KUKA KRL program: EPS_2_251825_SA36_A_20260116064122.src

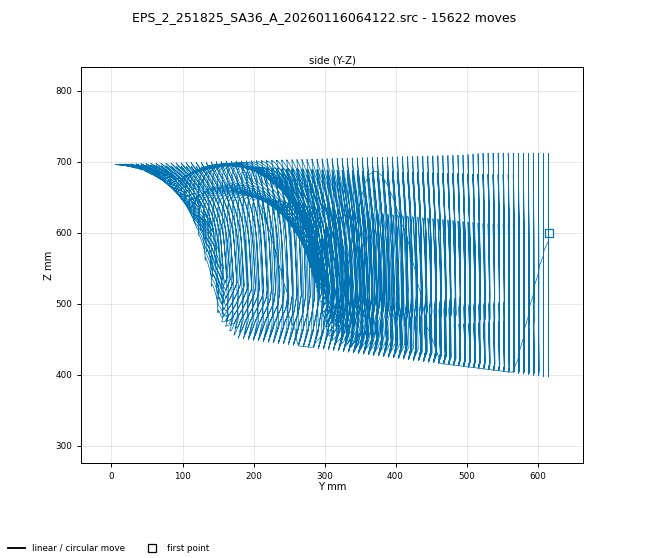
[picture p0: tool path of EPS_2_251825_SA36_A_20260116064122.src, 15622 of 15624 moves have a stored position in this frame; points joined in program order, loops and branches not executed]
&ACCESS RVP
&REL 4
&COMMENT QRS 19112012
&PARAM EDITMASK = *
DEF PART()
EXT BAS (BAS_COMMAND :IN,REAL :IN )
INT I
BAS (#INITMOV,0 )

;KUKA QRS Post kuka4.cps  Date:22-06-2017 !

File_ID=2974

QRS_PRE_INIT()

;Init var - Until changes are made in qrs_pre_init
Outlet_Square_prg=0
Inlet_1_Square_prg=0
Inlet_2_Square_prg=0
Inlet_3_Square_prg=0
Inlet_4_Square_prg=0
Inlet_5_Square_prg=0

Outlet_1={X 0.000, Y 524.580, Z 611.500, B 0.000, E1 0.000 }
Inlet_1={X 0.000, Y 531.710, Z 511.500, B 0.000, E1 90.000 }
Inlet_2={X 0.000, Y 526.720, Z 581.500, B 0.000, E1 180.000 }
Inlet_3={X 0.000, Y 526.720, Z 581.500, B 0.000, E1 270.000 }
Outlet_1_type=201
Inlet_1_type=201
Inlet_2_type=201
Inlet_3_type=201
;QRS#1=Sidecore dimensions
;QRS#2=200-8" PVC SDR 35
;QRS#3=200-8" PVC SDR 35
;QRS#4=200-8" PVC SDR 35
;QRS#5=200-8" PVC SDR 35
;QRS#6=
;QRS#7=
;QRS#8=
;QRS#9=12-08 PSX
;QRS#10=12-08 PSX
;QRS#11=12-08 PSX
;QRS#12=12-08 PSX
;QRS#13=
;QRS#14=
;QRS#15=
;QRS#16=1220x127x991 3,25'
;QRS#17=EPS Height
;QRS#18=712
;QRS#19=*
;QRS#20= UPDATED VERSION 22-06-2017
;QRS#21=*
Outlet_Square=0100
Inlet_1_Square=0100
Inlet_2_Square=0100
Inlet_3_Square=0100
Inlet_4_Square=0
Inlet_5_Square=0
Mill_Square=1
Outlet_Square_Prg=204
Inlet_1_Square_prg=204
Inlet_2_Square_prg=204
Inlet_3_Square_prg=204

QRS_INIT()

$ADVANCE=5

; T1
PTP {E1 173.498,E2 173.498}
PTP {X 0,Y 615.498,A -85,B 0,C 180,E1 173.498,E2 173.498,E3 0,E4 0,E5 0,E6 0}
QRS_SPEED_INIT()
LIN {X 0,Y 615.498,Z 600,A -85,B 0,C 180,E1 173.498,E2 173.498,E3 0,E4 0,E5 0,E6 0} C_VEL
LIN {X 0,Y 615.498,Z 591.852,A -85,B 0,C 180,E1 173.498,E2 173.498} C_VEL
LIN {X 0,Y 615.496,Z 590.208,A -85,B 0,C 180,E1 173.418,E2 173.418} C_VEL
LIN {X 0,Y 615.497,Z 582.536,A -85,B 0,C 180,E1 172.455,E2 172.455} C_VEL
LIN {X 0,Y 615.498,Z 572.758,A -85,B 0,C 180,E1 171.463,E2 171.463} C_VEL
LIN {X 0,Y 615.498,Z 562.492,A -85,B 0,C 180,E1 170.636,E2 170.636} C_VEL
LIN {X 0,Y 615.491,Z 550.929,A -85,B 0,C 180,E1 169.889,E2 169.889} C_VEL
LIN {X 0,Y 615.495,Z 539.071,A -85,B 0,C 180,E1 169.293,E2 169.293} C_VEL
LIN {X 0,Y 615.478,Z 526.159,A -85,B 0,C 180,E1 168.807,E2 168.807} C_VEL
LIN {X 0,Y 615.485,Z 513.556,A -85,B 0,C 180,E1 168.473,E2 168.473} C_VEL
LIN {X 0,Y 615.495,Z 500.425,A -85,B 0,C 180,E1 168.265,E2 168.265} C_VEL
LIN {X 0,Y 615.485,Z 402.646,A -85,B 0,C 180,E1 167.113,E2 167.113} C_VEL
LIN {X 0,Y 615.478,Z 396.69,A -85,B 0,C 180,E1 165.834,E2 165.834} C_VEL
LIN {X 0,Y 615.447,Z 396.692,A -85,B 0,C 180,E1 163.412,E2 163.412} C_VEL
LIN {X 0,Y 615.448,Z 396.692,A -85,B 0,C 180,E1 161.353,E2 161.353} C_VEL
LIN {X 0,Y 615.498,Z 396.7,A -85,B 0,C 180,E1 158.568,E2 158.568} C_VEL
LIN {X 0,Y 615.473,Z 396.686,A -85,B 0,C 180,E1 155.727,E2 155.727} C_VEL
LIN {X 0,Y 615.476,Z 396.697,A -85,B 0,C 180,E1 152.958,E2 152.958} C_VEL
LIN {X 0,Y 615.489,Z 396.686,A -85,B 0,C 180,E1 150.206,E2 150.206} C_VEL
LIN {X 0,Y 615.471,Z 396.688,A -85,B 0,C 180,E1 147.541,E2 147.541} C_VEL
LIN {X 0,Y 615.476,Z 396.696,A -85,B 0,C 180,E1 145.184,E2 145.184} C_VEL
LIN {X 0,Y 615.485,Z 396.696,A -85,B 0,C 180,E1 142.757,E2 142.757} C_VEL
LIN {X 0,Y 615.493,Z 396.682,A -85,B 0,C 180,E1 139.911,E2 139.911} C_VEL
LIN {X 0,Y 615.484,Z 396.697,A -85,B 0,C 180,E1 136.953,E2 136.953} C_VEL
LIN {X 0,Y 615.487,Z 396.684,A -85,B 0,C 180,E1 133.997,E2 133.997} C_VEL
LIN {X 0,Y 615.477,Z 396.698,A -85,B 0,C 180,E1 131.093,E2 131.093} C_VEL
LIN {X 0,Y 615.463,Z 396.694,A -85,B 0,C 180,E1 128.906,E2 128.906} C_VEL
LIN {X 0,Y 615.461,Z 396.689,A -85,B 0,C 180,E1 126.427,E2 126.427} C_VEL
LIN {X 0,Y 615.498,Z 396.699,A -85,B 0,C 180,E1 123.535,E2 123.535} C_VEL
LIN {X 0,Y 615.445,Z 396.695,A -85,B 0,C 180,E1 120.922,E2 120.922} C_VEL
LIN {X 0,Y 615.452,Z 396.692,A -85,B 0,C 180,E1 118.444,E2 118.444} C_VEL
LIN {X 0,Y 615.477,Z 396.7,A -85,B 0,C 180,E1 115.566,E2 115.566} C_VEL
LIN {X 0,Y 615.47,Z 396.699,A -85,B 0,C 180,E1 113.557,E2 113.557} C_VEL
LIN {X 0,Y 615.44,Z 396.801,A -85,B 0,C 180,E1 112.513,E2 112.513} C_VEL
LIN {X 0,Y 615.481,Z 417.648,A -85,B 0,C 180,E1 109.685,E2 109.685} C_VEL
LIN {X 0,Y 615.457,Z 437.029,A -85,B 0,C 180,E1 107.1,E2 107.1} C_VEL
LIN {X 0,Y 615.482,Z 457.56,A -85,B 0,C 180,E1 104.396,E2 104.396} C_VEL
LIN {X 0,Y 615.455,Z 469.845,A -85,B 0,C 180,E1 102.824,E2 102.824} C_VEL
LIN {X 0,Y 615.464,Z 577.646,A -85,B 0,C 180,E1 101.548,E2 101.548} C_VEL
LIN {X 0,Y 615.46,Z 590.227,A -85,B 0,C 180,E1 101.277,E2 101.277} C_VEL
LIN {X 0,Y 615.48,Z 602.525,A -85,B 0,C 180,E1 100.883,E2 100.883} C_VEL
LIN {X 0,Y 615.489,Z 614.565,A -85,B 0,C 180,E1 100.361,E2 100.361} C_VEL
LIN {X 0,Y 615.491,Z 626.304,A -85,B 0,C 180,E1 99.696,E2 99.696} C_VEL
LIN {X 0,Y 615.499,Z 636.767,A -85,B 0,C 180,E1 98.95,E2 98.95} C_VEL
LIN {X 0,Y 615.498,Z 645.33,A -85,B 0,C 180,E1 98.206,E2 98.206} C_VEL
LIN {X 0,Y 615.497,Z 653.209,A -85,B 0,C 180,E1 97.38,E2 97.38} C_VEL
LIN {X 0,Y 615.497,Z 660.898,A -85,B 0,C 180,E1 96.392,E2 96.392} C_VEL
LIN {X 0,Y 615.497,Z 667.958,A -85,B 0,C 180,E1 95.241,E2 95.241} C_VEL
LIN {X 0,Y 615.494,Z 672.658,A -85,B 0,C 180,E1 94.256,E2 94.256} C_VEL
LIN {X 0,Y 615.494,Z 676.254,A -85,B 0,C 180,E1 93.273,E2 93.273} C_VEL
LIN {X 0,Y 615.496,Z 678.115,A -85,B 0,C 180,E1 92.618,E2 92.618} C_VEL
LIN {X 0,Y 615.499,Z 679.533,A -85,B 0,C 180,E1 91.963,E2 91.963} C_VEL
LIN {X 0,Y 615.496,Z 681.141,A -85,B 0,C 180,E1 90.654,E2 90.654} C_VEL
LIN {X 0,Y 615.495,Z 681.384,A -85,B 0,C 180,E1 90,E2 90} C_VEL
LIN {X 0,Y 615.495,Z 681.206,A -85,B 0,C 180,E1 89.346,E2 89.346} C_VEL
LIN {X 0,Y 615.499,Z 679.682,A -85,B 0,C 180,E1 88.037,E2 88.037} C_VEL
LIN {X 0,Y 615.498,Z 678.341,A -85,B 0,C 180,E1 87.382,E2 87.382} C_VEL
LIN {X 0,Y 615.496,Z 675.494,A -85,B 0,C 180,E1 86.399,E2 86.399} C_VEL
LIN {X 0,Y 615.498,Z 671.634,A -85,B 0,C 180,E1 85.416,E2 85.416} C_VEL
LIN {X 0,Y 615.498,Z 666.651,A -85,B 0,C 180,E1 84.43,E2 84.43} C_VEL
LIN {X 0,Y 615.496,Z 660.208,A -85,B 0,C 180,E1 83.418,E2 83.418} C_VEL
LIN {X 0,Y 615.497,Z 652.536,A -85,B 0,C 180,E1 82.455,E2 82.455} C_VEL
LIN {X 0,Y 615.498,Z 642.758,A -85,B 0,C 180,E1 81.463,E2 81.463} C_VEL
LIN {X 0,Y 615.498,Z 632.492,A -85,B 0,C 180,E1 80.636,E2 80.636} C_VEL
LIN {X 0,Y 615.491,Z 620.929,A -85,B 0,C 180,E1 79.889,E2 79.889} C_VEL
LIN {X 0,Y 615.495,Z 609.089,A -85,B 0,C 180,E1 79.294,E2 79.294} C_VEL
LIN {X 0,Y 615.467,Z 596.161,A -85,B 0,C 180,E1 78.806,E2 78.806} C_VEL
LIN {X 0,Y 615.466,Z 583.56,A -85,B 0,C 180,E1 78.473,E2 78.473} C_VEL
LIN {X 0,Y 615.476,Z 570.434,A -85,B 0,C 180,E1 78.264,E2 78.264} C_VEL
LIN {X 0,Y 615.455,Z 469.493,A -85,B 0,C 180,E1 77.071,E2 77.071} C_VEL
LIN {X 0,Y 615.473,Z 449.33,A -85,B 0,C 180,E1 74.434,E2 74.434} C_VEL
LIN {X 0,Y 615.472,Z 427.636,A -85,B 0,C 180,E1 71.562,E2 71.562} C_VEL
LIN {X 0,Y 615.457,Z 407.969,A -85,B 0,C 180,E1 68.918,E2 68.918} C_VEL
LIN {X 0,Y 615.43,Z 396.698,A -85,B 0,C 180,E1 67.376,E2 67.376} C_VEL
LIN {X 0,Y 615.429,Z 396.697,A -85,B 0,C 180,E1 65.006,E2 65.006} C_VEL
LIN {X 0,Y 615.491,Z 396.694,A -85,B 0,C 180,E1 62.085,E2 62.085} C_VEL
LIN {X 0,Y 615.479,Z 396.689,A -85,B 0,C 180,E1 59.839,E2 59.839} C_VEL
LIN {X 0,Y 615.457,Z 396.69,A -85,B 0,C 180,E1 57.541,E2 57.541} C_VEL
LIN {X 0,Y 615.455,Z 396.694,A -85,B 0,C 180,E1 55.183,E2 55.183} C_VEL
LIN {X 0,Y 615.481,Z 396.701,A -85,B 0,C 180,E1 52.757,E2 52.757} C_VEL
LIN {X 0,Y 615.491,Z 396.683,A -85,B 0,C 180,E1 49.911,E2 49.911} C_VEL
LIN {X 0,Y 615.475,Z 396.687,A -85,B 0,C 180,E1 47.646,E2 47.646} C_VEL
LIN {X 0,Y 615.496,Z 396.7,A -85,B 0,C 180,E1 44.932,E2 44.932} C_VEL
LIN {X 0,Y 615.49,Z 396.683,A -85,B 0,C 180,E1 42.08,E2 42.08} C_VEL
LIN {X 0,Y 615.489,Z 396.698,A -85,B 0,C 180,E1 39.062,E2 39.062} C_VEL
LIN {X 0,Y 615.468,Z 396.688,A -85,B 0,C 180,E1 36.426,E2 36.426} C_VEL
LIN {X 0,Y 615.49,Z 396.697,A -85,B 0,C 180,E1 33.534,E2 33.534} C_VEL
LIN {X 0,Y 615.454,Z 396.695,A -85,B 0,C 180,E1 30.922,E2 30.922} C_VEL
LIN {X 0,Y 615.455,Z 396.691,A -85,B 0,C 180,E1 28.444,E2 28.444} C_VEL
LIN {X 0,Y 615.484,Z 396.7,A -85,B 0,C 180,E1 25.567,E2 25.567} C_VEL
LIN {X 0,Y 615.473,Z 396.699,A -85,B 0,C 180,E1 23.557,E2 23.557} C_VEL
LIN {X 0,Y 615.441,Z 396.801,A -85,B 0,C 180,E1 22.513,E2 22.513} C_VEL
LIN {X 0,Y 615.481,Z 417.648,A -85,B 0,C 180,E1 19.685,E2 19.685} C_VEL
LIN {X 0,Y 615.457,Z 437.029,A -85,B 0,C 180,E1 17.1,E2 17.1} C_VEL
LIN {X 0,Y 615.482,Z 457.56,A -85,B 0,C 180,E1 14.396,E2 14.396} C_VEL
LIN {X 0,Y 615.455,Z 469.843,A -85,B 0,C 180,E1 12.824,E2 12.824} C_VEL
LIN {X 0,Y 615.464,Z 577.645,A -85,B 0,C 180,E1 11.548,E2 11.548} C_VEL
LIN {X 0,Y 615.46,Z 590.226,A -85,B 0,C 180,E1 11.277,E2 11.277} C_VEL
LIN {X 0,Y 615.48,Z 602.525,A -85,B 0,C 180,E1 10.883,E2 10.883} C_VEL
LIN {X 0,Y 615.489,Z 614.564,A -85,B 0,C 180,E1 10.361,E2 10.361} C_VEL
LIN {X 0,Y 615.491,Z 626.303,A -85,B 0,C 180,E1 9.696,E2 9.696} C_VEL
LIN {X 0,Y 615.499,Z 636.767,A -85,B 0,C 180,E1 8.95,E2 8.95} C_VEL
LIN {X 0,Y 615.498,Z 645.33,A -85,B 0,C 180,E1 8.206,E2 8.206} C_VEL
LIN {X 0,Y 615.497,Z 653.209,A -85,B 0,C 180,E1 7.381,E2 7.381} C_VEL
LIN {X 0,Y 615.497,Z 660.898,A -85,B 0,C 180,E1 6.392,E2 6.392} C_VEL
LIN {X 0,Y 615.497,Z 667.958,A -85,B 0,C 180,E1 5.241,E2 5.241} C_VEL
LIN {X 0,Y 615.494,Z 672.658,A -85,B 0,C 180,E1 4.256,E2 4.256} C_VEL
LIN {X 0,Y 615.494,Z 676.254,A -85,B 0,C 180,E1 3.273,E2 3.273} C_VEL
LIN {X 0,Y 615.496,Z 678.115,A -85,B 0,C 180,E1 2.618,E2 2.618} C_VEL
LIN {X 0,Y 615.499,Z 679.533,A -85,B 0,C 180,E1 1.963,E2 1.963} C_VEL
LIN {X 0,Y 615.496,Z 681.141,A -85,B 0,C 180,E1 0.654,E2 0.654} C_VEL
LIN {X 0,Y 615.495,Z 681.384,A -85,B 0,C 180,E1 0,E2 0} C_VEL
LIN {X 0,Y 615.495,Z 681.206,A -85,B 0,C 180,E1 -0.654,E2 -0.654} C_VEL
LIN {X 0,Y 615.499,Z 679.682,A -85,B 0,C 180,E1 -1.963,E2 -1.963} C_VEL
LIN {X 0,Y 615.498,Z 678.341,A -85,B 0,C 180,E1 -2.618,E2 -2.618} C_VEL
LIN {X 0,Y 615.496,Z 675.494,A -85,B 0,C 180,E1 -3.601,E2 -3.601} C_VEL
LIN {X 0,Y 615.498,Z 671.634,A -85,B 0,C 180,E1 -4.584,E2 -4.584} C_VEL
LIN {X 0,Y 615.498,Z 666.651,A -85,B 0,C 180,E1 -5.57,E2 -5.57} C_VEL
LIN {X 0,Y 615.496,Z 660.208,A -85,B 0,C 180,E1 -6.582,E2 -6.582} C_VEL
LIN {X 0,Y 615.497,Z 652.537,A -85,B 0,C 180,E1 -7.545,E2 -7.545} C_VEL
LIN {X 0,Y 615.498,Z 642.759,A -85,B 0,C 180,E1 -8.536,E2 -8.536} C_VEL
LIN {X 0,Y 615.498,Z 632.493,A -85,B 0,C 180,E1 -9.364,E2 -9.364} C_VEL
LIN {X 0,Y 615.491,Z 620.93,A -85,B 0,C 180,E1 -10.111,E2 -10.111} C_VEL
LIN {X 0,Y 615.495,Z 609.09,A -85,B 0,C 180,E1 -10.706,E2 -10.706} C_VEL
LIN {X 0,Y 615.467,Z 596.163,A -85,B 0,C 180,E1 -11.193,E2 -11.193} C_VEL
LIN {X 0,Y 615.466,Z 583.562,A -85,B 0,C 180,E1 -11.527,E2 -11.527} C_VEL
LIN {X 0,Y 615.476,Z 570.437,A -85,B 0,C 180,E1 -11.736,E2 -11.736} C_VEL
LIN {X 0,Y 615.455,Z 469.493,A -85,B 0,C 180,E1 -12.929,E2 -12.929} C_VEL
LIN {X 0,Y 615.473,Z 449.33,A -85,B 0,C 180,E1 -15.566,E2 -15.566} C_VEL
LIN {X 0,Y 615.472,Z 427.636,A -85,B 0,C 180,E1 -18.438,E2 -18.438} C_VEL
LIN {X 0,Y 615.457,Z 407.969,A -85,B 0,C 180,E1 -21.082,E2 -21.082} C_VEL
LIN {X 0,Y 615.43,Z 396.698,A -85,B 0,C 180,E1 -22.624,E2 -22.624} C_VEL
LIN {X 0,Y 615.429,Z 396.697,A -85,B 0,C 180,E1 -24.994,E2 -24.994} C_VEL
LIN {X 0,Y 615.491,Z 396.694,A -85,B 0,C 180,E1 -27.915,E2 -27.915} C_VEL
LIN {X 0,Y 615.48,Z 396.689,A -85,B 0,C 180,E1 -30.161,E2 -30.161} C_VEL
LIN {X 0,Y 615.457,Z 396.69,A -85,B 0,C 180,E1 -32.459,E2 -32.459} C_VEL
LIN {X 0,Y 615.457,Z 396.694,A -85,B 0,C 180,E1 -34.817,E2 -34.817} C_VEL
LIN {X 0,Y 615.486,Z 396.701,A -85,B 0,C 180,E1 -37.242,E2 -37.242} C_VEL
LIN {X 0,Y 615.491,Z 396.683,A -85,B 0,C 180,E1 -40.089,E2 -40.089} C_VEL
LIN {X 0,Y 615.486,Z 396.702,A -85,B 0,C 180,E1 -43.047,E2 -43.047} C_VEL
LIN {X 0,Y 615.487,Z 396.683,A -85,B 0,C 180,E1 -46.003,E2 -46.003} C_VEL
LIN {X 0,Y 615.485,Z 396.702,A -85,B 0,C 180,E1 -48.906,E2 -48.906} C_VEL
LIN {X 0,Y 615.474,Z 396.695,A -85,B 0,C 180,E1 -51.094,E2 -51.094} C_VEL
LIN {X 0,Y 615.466,Z 396.688,A -85,B 0,C 180,E1 -53.574,E2 -53.574} C_VEL
LIN {X 0,Y 615.495,Z 396.697,A -85,B 0,C 180,E1 -56.465,E2 -56.465} C_VEL
LIN {X 0,Y 615.449,Z 396.695,A -85,B 0,C 180,E1 -59.078,E2 -59.078} C_VEL
LIN {X 0,Y 615.453,Z 396.692,A -85,B 0,C 180,E1 -61.556,E2 -61.556} C_VEL
LIN {X 0,Y 615.475,Z 396.699,A -85,B 0,C 180,E1 -64.434,E2 -64.434} C_VEL
LIN {X 0,Y 615.437,Z 396.843,A -85,B 0,C 180,E1 -65.411,E2 -65.411} C_VEL
LIN {X 0,Y 615.475,Z 420.552,A -85,B 0,C 180,E1 -68.216,E2 -68.216} C_VEL
LIN {X 0,Y 615.476,Z 443.127,A -85,B 0,C 180,E1 -70.835,E2 -70.835} C_VEL
LIN {X 0,Y 615.465,Z 467.126,A -85,B 0,C 180,E1 -73.577,E2 -73.577} C_VEL
LIN {X 0,Y 615.45,Z 492.711,A -85,B 0,C 180,E1 -76.462,E2 -76.462} C_VEL
LIN {X 0,Y 615.446,Z 498.522,A -85,B 0,C 180,E1 -77.113,E2 -77.113} C_VEL
LIN {X 0,Y 615.467,Z 607.831,A -85,B 0,C 180,E1 -78.41,E2 -78.41} C_VEL
LIN {X 0,Y 615.463,Z 620.346,A -85,B 0,C 180,E1 -78.681,E2 -78.681} C_VEL
LIN {X 0,Y 615.484,Z 633.665,A -85,B 0,C 180,E1 -79.115,E2 -79.115} C_VEL
LIN {X 0,Y 615.486,Z 645.476,A -85,B 0,C 180,E1 -79.639,E2 -79.639} C_VEL
LIN {X 0,Y 615.492,Z 656.993,A -85,B 0,C 180,E1 -80.304,E2 -80.304} C_VEL
LIN {X 0,Y 615.499,Z 667.34,A -85,B 0,C 180,E1 -81.05,E2 -81.05} C_VEL
LIN {X 0,Y 615.497,Z 675.811,A -85,B 0,C 180,E1 -81.794,E2 -81.794} C_VEL
LIN {X 0,Y 615.498,Z 683.606,A -85,B 0,C 180,E1 -82.62,E2 -82.62} C_VEL
LIN {X 0,Y 615.496,Z 691.203,A -85,B 0,C 180,E1 -83.608,E2 -83.608} C_VEL
LIN {X 0,Y 615.498,Z 698.204,A -85,B 0,C 180,E1 -84.759,E2 -84.759} C_VEL
LIN {X 0,Y 615.494,Z 702.851,A -85,B 0,C 180,E1 -85.744,E2 -85.744} C_VEL
LIN {X 0,Y 615.494,Z 706.399,A -85,B 0,C 180,E1 -86.727,E2 -86.727} C_VEL
LIN {X 0,Y 615.497,Z 708.233,A -85,B 0,C 180,E1 -87.382,E2 -87.382} C_VEL
LIN {X 0,Y 615.499,Z 709.608,A -85,B 0,C 180,E1 -88.037,E2 -88.037} C_VEL
LIN {X 0,Y 615.496,Z 711.174,A -85,B 0,C 180,E1 -89.346,E2 -89.346} C_VEL
LIN {X 0,Y 615.494,Z 711.389,A -85,B 0,C 180,E1 -90,E2 -90} C_VEL
LIN {X 0,Y 615.495,Z 710.58,A -85,B 0,C 180,E1 -91.309,E2 -91.309} C_VEL
LIN {X 0,Y 615.499,Z 709.608,A -85,B 0,C 180,E1 -91.963,E2 -91.963} C_VEL
LIN {X 0,Y 615.497,Z 708.233,A -85,B 0,C 180,E1 -92.618,E2 -92.618} C_VEL
LIN {X 0,Y 615.496,Z 705.349,A -85,B 0,C 180,E1 -93.601,E2 -93.601} C_VEL
LIN {X 0,Y 615.498,Z 701.441,A -85,B 0,C 180,E1 -94.584,E2 -94.584} C_VEL
LIN {X 0,Y 615.499,Z 696.405,A -85,B 0,C 180,E1 -95.57,E2 -95.57} C_VEL
LIN {X 0,Y 615.497,Z 689.869,A -85,B 0,C 180,E1 -96.583,E2 -96.583} C_VEL
LIN {X 0,Y 615.497,Z 682.133,A -85,B 0,C 180,E1 -97.545,E2 -97.545} C_VEL
LIN {X 0,Y 615.498,Z 674.044,A -85,B 0,C 180,E1 -98.371,E2 -98.371} C_VEL
LIN {X 0,Y 615.499,Z 664.167,A -85,B 0,C 180,E1 -99.199,E2 -99.199} C_VEL
LIN {X 0,Y 615.491,Z 652.98,A -85,B 0,C 180,E1 -99.945,E2 -99.945} C_VEL
LIN {X 0,Y 615.487,Z 642.021,A -85,B 0,C 180,E1 -100.527,E2 -100.527} C_VEL
LIN {X 0,Y 615.473,Z 629.516,A -85,B 0,C 180,E1 -101.039,E2 -101.039} C_VEL
LIN {X 0,Y 615.463,Z 617.067,A -85,B 0,C 180,E1 -101.402,E2 -101.402} C_VEL
LIN {X 0,Y 615.47,Z 603.466,A -85,B 0,C 180,E1 -101.652,E2 -101.652} C_VEL
LIN {X 0,Y 615.446,Z 498.522,A -85,B 0,C 180,E1 -102.887,E2 -102.887} C_VEL
LIN {X 0,Y 615.482,Z 474.694,A -85,B 0,C 180,E1 -105.566,E2 -105.566} C_VEL
LIN {X 0,Y 615.484,Z 450.837,A -85,B 0,C 180,E1 -108.28,E2 -108.28} C_VEL
LIN {X 0,Y 615.463,Z 428.078,A -85,B 0,C 180,E1 -110.907,E2 -110.907} C_VEL
LIN {X 0,Y 615.467,Z 405.498,A -85,B 0,C 180,E1 -113.557,E2 -113.557} C_VEL
LIN {X 0,Y 615.434,Z 396.696,A -85,B 0,C 180,E1 -114.634,E2 -114.634} C_VEL
LIN {X 0,Y 615.435,Z 396.697,A -85,B 0,C 180,E1 -117.035,E2 -117.035} C_VEL
LIN {X 0,Y 615.496,Z 396.696,A -85,B 0,C 180,E1 -119.796,E2 -119.796} C_VEL
LIN {X 0,Y 615.453,Z 396.691,A -85,B 0,C 180,E1 -122.46,E2 -122.46} C_VEL
LIN {X 0,Y 615.445,Z 396.694,A -85,B 0,C 180,E1 -124.818,E2 -124.818} C_VEL
LIN {X 0,Y 615.476,Z 396.698,A -85,B 0,C 180,E1 -127.243,E2 -127.243} C_VEL
LIN {X 0,Y 615.49,Z 396.684,A -85,B 0,C 180,E1 -130.089,E2 -130.089} C_VEL
LIN {X 0,Y 615.469,Z 396.687,A -85,B 0,C 180,E1 -132.355,E2 -132.355} C_VEL
LIN {X 0,Y 615.476,Z 396.699,A -85,B 0,C 180,E1 -135.07,E2 -135.07} C_VEL
LIN {X 0,Y 615.491,Z 396.683,A -85,B 0,C 180,E1 -137.92,E2 -137.92} C_VEL
LIN {X 0,Y 615.48,Z 396.685,A -85,B 0,C 180,E1 -140.249,E2 -140.249} C_VEL
LIN {X 0,Y 615.487,Z 396.702,A -85,B 0,C 180,E1 -143.064,E2 -143.064} C_VEL
LIN {X 0,Y 615.49,Z 396.682,A -85,B 0,C 180,E1 -145.978,E2 -145.978} C_VEL
LIN {X 0,Y 615.486,Z 396.703,A -85,B 0,C 180,E1 -148.915,E2 -148.915} C_VEL
LIN {X 0,Y 615.47,Z 396.688,A -85,B 0,C 180,E1 -151.553,E2 -151.553} C_VEL
LIN {X 0,Y 615.483,Z 396.69,A -85,B 0,C 180,E1 -154.284,E2 -154.284} C_VEL
LIN {X 0,Y 615.49,Z 396.694,A -85,B 0,C 180,E1 -156.444,E2 -156.444} C_VEL
LIN {X 0,Y 615.457,Z 396.692,A -85,B 0,C 180,E1 -159.268,E2 -159.268} C_VEL
LIN {X 0,Y 615.493,Z 396.686,A -85,B 0,C 180,E1 -162.043,E2 -162.043} C_VEL
LIN {X 0,Y 615.467,Z 396.697,A -85,B 0,C 180,E1 -164.773,E2 -164.773} C_VEL
LIN {X 0,Y 615.491,Z 396.874,A -85,B 0,C 180,E1 -165.988,E2 -165.988} C_VEL
LIN {X 0,Y 615.486,Z 402.617,A -85,B 0,C 180,E1 -167.197,E2 -167.197} C_VEL
LIN {X 0,Y 615.487,Z 508.791,A -85,B 0,C 180,E1 -168.473,E2 -168.473} C_VEL
LIN {X 0,Y 615.477,Z 521.741,A -85,B 0,C 180,E1 -168.765,E2 -168.765} C_VEL
LIN {X 0,Y 615.488,Z 533.654,A -85,B 0,C 180,E1 -169.159,E2 -169.159} C_VEL
LIN {X 0,Y 615.489,Z 546.195,A -85,B 0,C 180,E1 -169.723,E2 -169.723} C_VEL
LIN {X 0,Y 615.491,Z 557.576,A -85,B 0,C 180,E1 -170.387,E2 -170.387} C_VEL
LIN {X 0,Y 615.498,Z 567.823,A -85,B 0,C 180,E1 -171.133,E2 -171.133} C_VEL
LIN {X 0,Y 615.499,Z 577.034,A -85,B 0,C 180,E1 -171.959,E2 -171.959} C_VEL
LIN {X 0,Y 615.499,Z 585.892,A -85,B 0,C 180,E1 -172.943,E2 -172.943} C_VEL
LIN {X 0,Y 615.497,Z 593.123,A -85,B 0,C 180,E1 -173.937,E2 -173.937} C_VEL
LIN {X 0,Y 615.497,Z 597.958,A -85,B 0,C 180,E1 -174.759,E2 -174.759} C_VEL
LIN {X 0,Y 615.494,Z 602.658,A -85,B 0,C 180,E1 -175.744,E2 -175.744} C_VEL
LIN {X 0,Y 615.494,Z 606.255,A -85,B 0,C 180,E1 -176.727,E2 -176.727} C_VEL
LIN {X 0,Y 615.496,Z 608.115,A -85,B 0,C 180,E1 -177.382,E2 -177.382} C_VEL
LIN {X 0,Y 615.499,Z 609.533,A -85,B 0,C 180,E1 -178.037,E2 -178.037} C_VEL
LIN {X 0,Y 615.496,Z 611.142,A -85,B 0,C 180,E1 -179.346,E2 -179.346} C_VEL
LIN {X 0,Y 615.495,Z 611.384,A -85,B 0,C 180,E1 -180,E2 -180} C_VEL
LIN {X 0,Y 615.495,Z 611.206,A -85,B 0,C 180,E1 -180.654,E2 -180.654} C_VEL
LIN {X 0,Y 615.499,Z 609.682,A -85,B 0,C 180,E1 -181.963,E2 -181.963} C_VEL
LIN {X 0,Y 615.498,Z 608.341,A -85,B 0,C 180,E1 -182.618,E2 -182.618} C_VEL
LIN {X 0,Y 615.496,Z 605.494,A -85,B 0,C 180,E1 -183.601,E2 -183.601} C_VEL
LIN {X 0,Y 615.498,Z 601.634,A -85,B 0,C 180,E1 -184.585,E2 -184.585} C_VEL
LIN {X 0,Y 615.498,Z 596.651,A -85,B 0,C 180,E1 -185.57,E2 -185.57} C_VEL
LIN {X 0,Y 615.496,Z 590.208,A -85,B 0,C 180,E1 -186.582,E2 -186.582} C_VEL
LIN {X 0,Y 614.829,Z 587.026,A -85,B 0,C 180,E1 -187.031,E2 -187.031} C_VEL
LIN {X 0,Y 611.989,Z 581.452,A -85,B 0,C 180,E1 -187.748,E2 -187.748} C_VEL
LIN {X 0,Y 609.138,Z 575.177,A -85,B 0,C 180,E1 -188.429,E2 -188.429} C_VEL
LIN {X 0,Y 608.477,Z 570.935,A -85,B 0,C 180,E1 -188.819,E2 -188.819} C_VEL
LIN {X 0,Y 608.496,Z 560.383,A -85,B 0,C 180,E1 -189.641,E2 -189.641} C_VEL
LIN {X 0,Y 608.489,Z 549.612,A -85,B 0,C 180,E1 -190.313,E2 -190.313} C_VEL
LIN {X 0,Y 608.523,Z 536.856,A -85,B 0,C 180,E1 -190.932,E2 -190.932} C_VEL
LIN {X 0,Y 608.512,Z 524.956,A -85,B 0,C 180,E1 -191.365,E2 -191.365} C_VEL
LIN {X 0,Y 608.555,Z 512.656,A -85,B 0,C 180,E1 -191.681,E2 -191.681} C_VEL
LIN {X 0,Y 608.566,Z 496.956,A -85,B 0,C 180,E1 -191.913,E2 -191.913} C_VEL
LIN {X 0,Y 608.463,Z 402.885,A -85,B 0,C 180,E1 -193.038,E2 -193.038} C_VEL
LIN {X 0,Y 608.455,Z 397.69,A -85,B 0,C 180,E1 -194.166,E2 -194.166} C_VEL
LIN {X 0,Y 608.423,Z 397.692,A -85,B 0,C 180,E1 -196.785,E2 -196.785} C_VEL
LIN {X 0,Y 608.448,Z 397.698,A -85,B 0,C 180,E1 -199.571,E2 -199.571} C_VEL
LIN {X 0,Y 608.432,Z 397.69,A -85,B 0,C 180,E1 -202.469,E2 -202.469} C_VEL
LIN {X 0,Y 608.44,Z 397.69,A -85,B 0,C 180,E1 -204.572,E2 -204.572} C_VEL
LIN {X 0,Y 608.475,Z 397.694,A -85,B 0,C 180,E1 -207.206,E2 -207.206} C_VEL
LIN {X 0,Y 608.469,Z 397.686,A -85,B 0,C 180,E1 -209.971,E2 -209.971} C_VEL
LIN {X 0,Y 608.452,Z 397.694,A -85,B 0,C 180,E1 -212.88,E2 -212.88} C_VEL
LIN {X 0,Y 608.437,Z 397.696,A -85,B 0,C 180,E1 -215.278,E2 -215.278} C_VEL
LIN {X 0,Y 608.469,Z 397.686,A -85,B 0,C 180,E1 -217.747,E2 -217.747} C_VEL
LIN {X 0,Y 608.454,Z 397.689,A -85,B 0,C 180,E1 -220.329,E2 -220.329} C_VEL
LIN {X 0,Y 608.451,Z 397.697,A -85,B 0,C 180,E1 -222.96,E2 -222.96} C_VEL
LIN {X 0,Y 608.455,Z 397.687,A -85,B 0,C 180,E1 -225.737,E2 -225.737} C_VEL
LIN {X 0,Y 608.467,Z 397.686,A -85,B 0,C 180,E1 -227.939,E2 -227.939} C_VEL
LIN {X 0,Y 608.44,Z 397.699,A -85,B 0,C 180,E1 -230.706,E2 -230.706} C_VEL
LIN {X 0,Y 608.428,Z 397.693,A -85,B 0,C 180,E1 -233.083,E2 -233.083} C_VEL
LIN {X 0,Y 608.449,Z 397.688,A -85,B 0,C 180,E1 -235.529,E2 -235.529} C_VEL
LIN {X 0,Y 608.456,Z 397.689,A -85,B 0,C 180,E1 -237.905,E2 -237.905} C_VEL
LIN {X 0,Y 608.48,Z 397.692,A -85,B 0,C 180,E1 -240.221,E2 -240.221} C_VEL
LIN {X 0,Y 608.408,Z 397.693,A -85,B 0,C 180,E1 -243.224,E2 -243.224} C_VEL
LIN {X 0,Y 608.423,Z 397.692,A -85,B 0,C 180,E1 -245.428,E2 -245.428} C_VEL
LIN {X 0,Y 608.439,Z 397.85,A -85,B 0,C 180,E1 -247.358,E2 -247.358} C_VEL
LIN {X 0,Y 608.549,Z 411.949,A -85,B 0,C 180,E1 -249.302,E2 -249.302} C_VEL
LIN {X 0,Y 608.546,Z 433.194,A -85,B 0,C 180,E1 -252.179,E2 -252.179} C_VEL
LIN {X 0,Y 608.496,Z 455.195,A -85,B 0,C 180,E1 -255.109,E2 -255.109} C_VEL
LIN {X 0,Y 608.458,Z 469.921,A -85,B 0,C 180,E1 -257.026,E2 -257.026} C_VEL
LIN {X 0,Y 608.536,Z 577.771,A -85,B 0,C 180,E1 -258.319,E2 -258.319} C_VEL
LIN {X 0,Y 608.512,Z 591.118,A -85,B 0,C 180,E1 -258.614,E2 -258.614} C_VEL
LIN {X 0,Y 608.521,Z 604.463,A -85,B 0,C 180,E1 -259.059,E2 -259.059} C_VEL
LIN {X 0,Y 608.499,Z 616.36,A -85,B 0,C 180,E1 -259.603,E2 -259.603} C_VEL
LIN {X 0,Y 608.504,Z 627.785,A -85,B 0,C 180,E1 -260.275,E2 -260.275} C_VEL
LIN {X 0,Y 608.474,Z 638.082,A -85,B 0,C 180,E1 -261.029,E2 -261.029} C_VEL
LIN {X 0,Y 608.464,Z 647.35,A -85,B 0,C 180,E1 -261.866,E2 -261.866} C_VEL
LIN {X 0,Y 608.466,Z 656.323,A -85,B 0,C 180,E1 -262.867,E2 -262.867} C_VEL
LIN {X 0,Y 608.444,Z 663.553,A -85,B 0,C 180,E1 -263.867,E2 -263.867} C_VEL
LIN {X 0,Y 608.462,Z 668.433,A -85,B 0,C 180,E1 -264.698,E2 -264.698} C_VEL
LIN {X 0,Y 608.439,Z 673.176,A -85,B 0,C 180,E1 -265.694,E2 -265.694} C_VEL
LIN {X 0,Y 608.425,Z 676.811,A -85,B 0,C 180,E1 -266.689,E2 -266.689} C_VEL
LIN {X 0,Y 608.425,Z 678.691,A -85,B 0,C 180,E1 -267.352,E2 -267.352} C_VEL
LIN {X 0,Y 608.444,Z 680.127,A -85,B 0,C 180,E1 -268.014,E2 -268.014} C_VEL
LIN {X 0,Y 608.439,Z 681.752,A -85,B 0,C 180,E1 -269.338,E2 -269.338} C_VEL
LIN {X 0,Y 608.435,Z 681.995,A -85,B 0,C 180,E1 -270,E2 -270} C_VEL
LIN {X 0,Y 608.438,Z 681.815,A -85,B 0,C 180,E1 -270.662,E2 -270.662} C_VEL
LIN {X 0,Y 608.444,Z 680.276,A -85,B 0,C 180,E1 -271.986,E2 -271.986} C_VEL
LIN {X 0,Y 608.426,Z 678.917,A -85,B 0,C 180,E1 -272.648,E2 -272.648} C_VEL
LIN {X 0,Y 608.449,Z 676.041,A -85,B 0,C 180,E1 -273.642,E2 -273.642} C_VEL
LIN {X 0,Y 608.433,Z 672.141,A -85,B 0,C 180,E1 -274.638,E2 -274.638} C_VEL
LIN {X 0,Y 608.449,Z 667.111,A -85,B 0,C 180,E1 -275.634,E2 -275.634} C_VEL
LIN {X 0,Y 608.441,Z 660.795,A -85,B 0,C 180,E1 -276.633,E2 -276.633} C_VEL
LIN {X 0,Y 608.475,Z 652.878,A -85,B 0,C 180,E1 -277.633,E2 -277.633} C_VEL
LIN {X 0,Y 608.472,Z 643.031,A -85,B 0,C 180,E1 -278.636,E2 -278.636} C_VEL
LIN {X 0,Y 608.48,Z 632.714,A -85,B 0,C 180,E1 -279.473,E2 -279.473} C_VEL
LIN {X 0,Y 608.488,Z 621.101,A -85,B 0,C 180,E1 -280.229,E2 -280.229} C_VEL
LIN {X 0,Y 608.524,Z 609.907,A -85,B 0,C 180,E1 -280.801,E2 -280.801} C_VEL
LIN {X 0,Y 608.517,Z 597.255,A -85,B 0,C 180,E1 -281.29,E2 -281.29} C_VEL
LIN {X 0,Y 608.516,Z 584.552,A -85,B 0,C 180,E1 -281.64,E2 -281.64} C_VEL
LIN {X 0,Y 608.533,Z 572.285,A -85,B 0,C 180,E1 -281.85,E2 -281.85} C_VEL
LIN {X 0,Y 608.45,Z 469.632,A -85,B 0,C 180,E1 -283.081,E2 -283.081} C_VEL
LIN {X 0,Y 608.488,Z 449.401,A -85,B 0,C 180,E1 -285.749,E2 -285.749} C_VEL
LIN {X 0,Y 608.517,Z 428.863,A -85,B 0,C 180,E1 -288.494,E2 -288.494} C_VEL
LIN {X 0,Y 608.54,Z 409.262,A -85,B 0,C 180,E1 -291.156,E2 -291.156} C_VEL
LIN {X 0,Y 608.419,Z 397.694,A -85,B 0,C 180,E1 -292.766,E2 -292.766} C_VEL
LIN {X 0,Y 608.415,Z 397.696,A -85,B 0,C 180,E1 -295.303,E2 -295.303} C_VEL
LIN {X 0,Y 608.43,Z 397.692,A -85,B 0,C 180,E1 -298.268,E2 -298.268} C_VEL
LIN {X 0,Y 608.43,Z 397.691,A -85,B 0,C 180,E1 -300.547,E2 -300.547} C_VEL
LIN {X 0,Y 608.439,Z 397.691,A -85,B 0,C 180,E1 -302.881,E2 -302.881} C_VEL
LIN {X 0,Y 608.436,Z 397.698,A -85,B 0,C 180,E1 -305.278,E2 -305.278} C_VEL
LIN {X 0,Y 608.468,Z 397.689,A -85,B 0,C 180,E1 -307.747,E2 -307.747} C_VEL
LIN {X 0,Y 608.446,Z 397.689,A -85,B 0,C 180,E1 -310.328,E2 -310.328} C_VEL
LIN {X 0,Y 608.45,Z 397.696,A -85,B 0,C 180,E1 -312.96,E2 -312.96} C_VEL
LIN {X 0,Y 608.459,Z 397.688,A -85,B 0,C 180,E1 -315.736,E2 -315.736} C_VEL
LIN {X 0,Y 608.46,Z 397.693,A -85,B 0,C 180,E1 -318.658,E2 -318.658} C_VEL
LIN {X 0,Y 608.436,Z 397.692,A -85,B 0,C 180,E1 -321.409,E2 -321.409} C_VEL
LIN {X 0,Y 608.45,Z 397.689,A -85,B 0,C 180,E1 -323.955,E2 -323.955} C_VEL
LIN {X 0,Y 608.468,Z 397.691,A -85,B 0,C 180,E1 -326.329,E2 -326.329} C_VEL
LIN {X 0,Y 608.443,Z 397.696,A -85,B 0,C 180,E1 -328.734,E2 -328.734} C_VEL
LIN {X 0,Y 608.444,Z 397.689,A -85,B 0,C 180,E1 -331.386,E2 -331.386} C_VEL
LIN {X 0,Y 608.478,Z 397.695,A -85,B 0,C 180,E1 -334.279,E2 -334.279} C_VEL
LIN {X 0,Y 608.416,Z 397.695,A -85,B 0,C 180,E1 -336.875,E2 -336.875} C_VEL
LIN {X 0,Y 608.439,Z 397.85,A -85,B 0,C 180,E1 -337.358,E2 -337.358} C_VEL
LIN {X 0,Y 608.549,Z 411.948,A -85,B 0,C 180,E1 -339.302,E2 -339.302} C_VEL
LIN {X 0,Y 608.546,Z 433.193,A -85,B 0,C 180,E1 -342.179,E2 -342.179} C_VEL
LIN {X 0,Y 608.496,Z 455.194,A -85,B 0,C 180,E1 -345.109,E2 -345.109} C_VEL
LIN {X 0,Y 608.458,Z 469.919,A -85,B 0,C 180,E1 -347.026,E2 -347.026} C_VEL
LIN {X 0,Y 608.536,Z 577.776,A -85,B 0,C 180,E1 -348.319,E2 -348.319} C_VEL
LIN {X 0,Y 608.512,Z 591.119,A -85,B 0,C 180,E1 -348.614,E2 -348.614} C_VEL
LIN {X 0,Y 608.531,Z 603.329,A -85,B 0,C 180,E1 -349.016,E2 -349.016} C_VEL
LIN {X 0,Y 608.508,Z 614.733,A -85,B 0,C 180,E1 -349.519,E2 -349.519} C_VEL
LIN {X 0,Y 608.482,Z 626.513,A -85,B 0,C 180,E1 -350.191,E2 -350.191} C_VEL
LIN {X 0,Y 608.474,Z 638.084,A -85,B 0,C 180,E1 -351.029,E2 -351.029} C_VEL
LIN {X 0,Y 608.464,Z 647.347,A -85,B 0,C 180,E1 -351.866,E2 -351.866} C_VEL
LIN {X 0,Y 608.466,Z 656.322,A -85,B 0,C 180,E1 -352.867,E2 -352.867} C_VEL
LIN {X 0,Y 608.444,Z 663.555,A -85,B 0,C 180,E1 -353.866,E2 -353.866} C_VEL
LIN {X 0,Y 608.462,Z 668.435,A -85,B 0,C 180,E1 -354.698,E2 -354.698} C_VEL
LIN {X 0,Y 608.439,Z 673.179,A -85,B 0,C 180,E1 -355.694,E2 -355.694} C_VEL
LIN {X 0,Y 608.425,Z 676.813,A -85,B 0,C 180,E1 -356.689,E2 -356.689} C_VEL
LIN {X 0,Y 608.425,Z 678.69,A -85,B 0,C 180,E1 -357.352,E2 -357.352} C_VEL
LIN {X 0,Y 608.444,Z 680.126,A -85,B 0,C 180,E1 -358.014,E2 -358.014} C_VEL
LIN {X 0,Y 608.439,Z 681.752,A -85,B 0,C 180,E1 -359.338,E2 -359.338} C_VEL
LIN {X 0,Y 608.435,Z 681.995,A -85,B 0,C 180,E1 -360,E2 -360} C_VEL
LIN {X 0,Y 608.438,Z 681.815,A -85,B 0,C 180,E1 -360.662,E2 -360.662} C_VEL
LIN {X 0,Y 608.444,Z 680.276,A -85,B 0,C 180,E1 -361.986,E2 -361.986} C_VEL
LIN {X 0,Y 608.426,Z 678.919,A -85,B 0,C 180,E1 -362.648,E2 -362.648} C_VEL
LIN {X 0,Y 608.449,Z 676.042,A -85,B 0,C 180,E1 -363.642,E2 -363.642} C_VEL
LIN {X 0,Y 608.433,Z 672.143,A -85,B 0,C 180,E1 -364.638,E2 -364.638} C_VEL
LIN {X 0,Y 608.449,Z 667.112,A -85,B 0,C 180,E1 -365.634,E2 -365.634} C_VEL
LIN {X 0,Y 608.441,Z 660.791,A -85,B 0,C 180,E1 -366.633,E2 -366.633} C_VEL
LIN {X 0,Y 608.475,Z 652.879,A -85,B 0,C 180,E1 -367.633,E2 -367.633} C_VEL
LIN {X 0,Y 608.472,Z 643.036,A -85,B 0,C 180,E1 -368.636,E2 -368.636} C_VEL
LIN {X 0,Y 608.48,Z 632.709,A -85,B 0,C 180,E1 -369.473,E2 -369.473} C_VEL
LIN {X 0,Y 608.487,Z 621.097,A -85,B 0,C 180,E1 -370.229,E2 -370.229} C_VEL
LIN {X 0,Y 608.524,Z 609.914,A -85,B 0,C 180,E1 -370.801,E2 -370.801} C_VEL
LIN {X 0,Y 608.517,Z 597.252,A -85,B 0,C 180,E1 -371.29,E2 -371.29} C_VEL
LIN {X 0,Y 608.516,Z 584.55,A -85,B 0,C 180,E1 -371.64,E2 -371.64} C_VEL
LIN {X 0,Y 608.533,Z 572.288,A -85,B 0,C 180,E1 -371.85,E2 -371.85} C_VEL
LIN {X 0,Y 608.45,Z 469.632,A -85,B 0,C 180,E1 -373.081,E2 -373.081} C_VEL
LIN {X 0,Y 608.488,Z 449.402,A -85,B 0,C 180,E1 -375.749,E2 -375.749} C_VEL
LIN {X 0,Y 608.517,Z 428.863,A -85,B 0,C 180,E1 -378.494,E2 -378.494} C_VEL
LIN {X 0,Y 608.54,Z 409.263,A -85,B 0,C 180,E1 -381.156,E2 -381.156} C_VEL
LIN {X 0,Y 608.419,Z 397.694,A -85,B 0,C 180,E1 -382.766,E2 -382.766} C_VEL
LIN {X 0,Y 608.416,Z 397.696,A -85,B 0,C 180,E1 -385.303,E2 -385.303} C_VEL
LIN {X 0,Y 608.431,Z 397.692,A -85,B 0,C 180,E1 -388.268,E2 -388.268} C_VEL
LIN {X 0,Y 608.43,Z 397.691,A -85,B 0,C 180,E1 -390.547,E2 -390.547} C_VEL
LIN {X 0,Y 608.442,Z 397.691,A -85,B 0,C 180,E1 -392.881,E2 -392.881} C_VEL
LIN {X 0,Y 608.436,Z 397.698,A -85,B 0,C 180,E1 -395.278,E2 -395.278} C_VEL
LIN {X 0,Y 608.469,Z 397.689,A -85,B 0,C 180,E1 -397.746,E2 -397.746} C_VEL
LIN {X 0,Y 608.447,Z 397.689,A -85,B 0,C 180,E1 -400.328,E2 -400.328} C_VEL
LIN {X 0,Y 608.451,Z 397.696,A -85,B 0,C 180,E1 -402.96,E2 -402.96} C_VEL
LIN {X 0,Y 608.459,Z 397.688,A -85,B 0,C 180,E1 -405.736,E2 -405.736} C_VEL
LIN {X 0,Y 608.461,Z 397.694,A -85,B 0,C 180,E1 -408.658,E2 -408.658} C_VEL
LIN {X 0,Y 608.464,Z 397.686,A -85,B 0,C 180,E1 -411.76,E2 -411.76} C_VEL
LIN {X 0,Y 608.449,Z 397.689,A -85,B 0,C 180,E1 -413.955,E2 -413.955} C_VEL
LIN {X 0,Y 608.471,Z 397.692,A -85,B 0,C 180,E1 -416.33,E2 -416.33} C_VEL
LIN {X 0,Y 608.441,Z 397.695,A -85,B 0,C 180,E1 -418.734,E2 -418.734} C_VEL
LIN {X 0,Y 608.441,Z 397.689,A -85,B 0,C 180,E1 -421.386,E2 -421.386} C_VEL
LIN {X 0,Y 608.474,Z 397.695,A -85,B 0,C 180,E1 -424.279,E2 -424.279} C_VEL
LIN {X 0,Y 608.422,Z 397.784,A -85,B 0,C 180,E1 -425.223,E2 -425.223} C_VEL
LIN {X 0,Y 608.613,Z 407.004,A -85,B 0,C 180,E1 -426.342,E2 -426.342} C_VEL
LIN {X 0,Y 608.566,Z 428.078,A -85,B 0,C 180,E1 -428.845,E2 -428.845} C_VEL
LIN {X 0,Y 608.553,Z 452.258,A -85,B 0,C 180,E1 -431.668,E2 -431.668} C_VEL
LIN {X 0,Y 608.476,Z 477.754,A -85,B 0,C 180,E1 -434.594,E2 -434.594} C_VEL
LIN {X 0,Y 608.444,Z 498.64,A -85,B 0,C 180,E1 -436.962,E2 -436.962} C_VEL
LIN {X 0,Y 608.531,Z 607.943,A -85,B 0,C 180,E1 -438.276,E2 -438.276} C_VEL
LIN {X 0,Y 608.498,Z 621.214,A -85,B 0,C 180,E1 -438.571,E2 -438.571} C_VEL
LIN {X 0,Y 608.512,Z 633.646,A -85,B 0,C 180,E1 -438.983,E2 -438.983} C_VEL
LIN {X 0,Y 608.504,Z 645.634,A -85,B 0,C 180,E1 -439.519,E2 -439.519} C_VEL
LIN {X 0,Y 608.483,Z 657.196,A -85,B 0,C 180,E1 -440.191,E2 -440.191} C_VEL
LIN {X 0,Y 608.485,Z 667.593,A -85,B 0,C 180,E1 -440.946,E2 -440.946} C_VEL
LIN {X 0,Y 608.475,Z 676.111,A -85,B 0,C 180,E1 -441.699,E2 -441.699} C_VEL
LIN {X 0,Y 608.471,Z 683.96,A -85,B 0,C 180,E1 -442.534,E2 -442.534} C_VEL
LIN {X 0,Y 608.461,Z 691.286,A -85,B 0,C 180,E1 -443.484,E2 -443.484} C_VEL
LIN {X 0,Y 608.45,Z 696.866,A -85,B 0,C 180,E1 -444.366,E2 -444.366} C_VEL
LIN {X 0,Y 608.432,Z 701.95,A -85,B 0,C 180,E1 -445.362,E2 -445.362} C_VEL
LIN {X 0,Y 608.449,Z 705.896,A -85,B 0,C 180,E1 -446.358,E2 -446.358} C_VEL
LIN {X 0,Y 608.425,Z 708.809,A -85,B 0,C 180,E1 -447.352,E2 -447.352} C_VEL
LIN {X 0,Y 608.444,Z 710.201,A -85,B 0,C 180,E1 -448.014,E2 -448.014} C_VEL
LIN {X 0,Y 608.438,Z 711.783,A -85,B 0,C 180,E1 -449.338,E2 -449.338} C_VEL
LIN {X 0,Y 608.434,Z 712,A -85,B 0,C 180,E1 -450,E2 -450} C_VEL
LIN {X 0,Y 608.448,Z 711.184,A -85,B 0,C 180,E1 -451.324,E2 -451.324} C_VEL
LIN {X 0,Y 608.444,Z 710.201,A -85,B 0,C 180,E1 -451.986,E2 -451.986} C_VEL
LIN {X 0,Y 608.425,Z 708.809,A -85,B 0,C 180,E1 -452.648,E2 -452.648} C_VEL
LIN {X 0,Y 608.449,Z 705.896,A -85,B 0,C 180,E1 -453.642,E2 -453.642} C_VEL
LIN {X 0,Y 608.432,Z 701.95,A -85,B 0,C 180,E1 -454.638,E2 -454.638} C_VEL
LIN {X 0,Y 608.437,Z 695.876,A -85,B 0,C 180,E1 -455.801,E2 -455.801} C_VEL
LIN {X 0,Y 608.462,Z 689.235,A -85,B 0,C 180,E1 -456.799,E2 -456.799} C_VEL
LIN {X 0,Y 608.456,Z 680.989,A -85,B 0,C 180,E1 -457.8,E2 -457.8} C_VEL
LIN {X 0,Y 608.472,Z 672.536,A -85,B 0,C 180,E1 -458.636,E2 -458.636} C_VEL
LIN {X 0,Y 608.478,Z 662.09,A -85,B 0,C 180,E1 -459.473,E2 -459.473} C_VEL
LIN {X 0,Y 608.501,Z 651.755,A -85,B 0,C 180,E1 -460.145,E2 -460.145} C_VEL
LIN {X 0,Y 608.517,Z 640.6,A -85,B 0,C 180,E1 -460.724,E2 -460.724} C_VEL
LIN {X 0,Y 608.515,Z 628.899,A -85,B 0,C 180,E1 -461.192,E2 -461.192} C_VEL
LIN {X 0,Y 608.528,Z 616.264,A -85,B 0,C 180,E1 -461.555,E2 -461.555} C_VEL
LIN {X 0,Y 608.533,Z 603.597,A -85,B 0,C 180,E1 -461.787,E2 -461.787} C_VEL
LIN {X 0,Y 608.46,Z 498.64,A -85,B 0,C 180,E1 -463.038,E2 -463.038} C_VEL
LIN {X 0,Y 608.536,Z 473.238,A -85,B 0,C 180,E1 -465.92,E2 -465.92} C_VEL
LIN {X 0,Y 608.562,Z 448.729,A -85,B 0,C 180,E1 -468.741,E2 -468.741} C_VEL
LIN {X 0,Y 608.552,Z 426.573,A -85,B 0,C 180,E1 -471.333,E2 -471.333} C_VEL
LIN {X 0,Y 608.642,Z 405.498,A -85,B 0,C 180,E1 -473.838,E2 -473.838} C_VEL
LIN {X 0,Y 608.42,Z 397.784,A -85,B 0,C 180,E1 -474.777,E2 -474.777} C_VEL
LIN {X 0,Y 608.421,Z 397.694,A -85,B 0,C 180,E1 -477.196,E2 -477.196} C_VEL
LIN {X 0,Y 608.471,Z 397.691,A -85,B 0,C 180,E1 -479.972,E2 -479.972} C_VEL
LIN {X 0,Y 608.435,Z 397.691,A -85,B 0,C 180,E1 -482.881,E2 -482.881} C_VEL
LIN {X 0,Y 608.434,Z 397.696,A -85,B 0,C 180,E1 -485.278,E2 -485.278} C_VEL
LIN {X 0,Y 608.462,Z 397.687,A -85,B 0,C 180,E1 -488.239,E2 -488.239} C_VEL
LIN {X 0,Y 608.462,Z 397.697,A -85,B 0,C 180,E1 -491.342,E2 -491.342} C_VEL
LIN {X 0,Y 608.454,Z 397.687,A -85,B 0,C 180,E1 -494.263,E2 -494.263} C_VEL
LIN {X 0,Y 608.445,Z 397.696,A -85,B 0,C 180,E1 -497.039,E2 -497.039} C_VEL
LIN {X 0,Y 608.456,Z 397.689,A -85,B 0,C 180,E1 -499.697,E2 -499.697} C_VEL
LIN {X 0,Y 608.466,Z 397.686,A -85,B 0,C 180,E1 -502.253,E2 -502.253} C_VEL
LIN {X 0,Y 608.45,Z 397.697,A -85,B 0,C 180,E1 -505.095,E2 -505.095} C_VEL
LIN {X 0,Y 608.46,Z 397.687,A -85,B 0,C 180,E1 -507.905,E2 -507.905} C_VEL
LIN {X 0,Y 608.472,Z 397.687,A -85,B 0,C 180,E1 -510.221,E2 -510.221} C_VEL
LIN {X 0,Y 608.44,Z 397.693,A -85,B 0,C 180,E1 -513.225,E2 -513.225} C_VEL
LIN {X 0,Y 608.481,Z 397.684,A -85,B 0,C 180,E1 -515.848,E2 -515.848} C_VEL
LIN {X 0,Y 608.474,Z 397.69,A -85,B 0,C 180,E1 -518.309,E2 -518.309} C_VEL
LIN {X 0,Y 608.444,Z 397.691,A -85,B 0,C 180,E1 -521.13,E2 -521.13} C_VEL
LIN {X 0,Y 608.456,Z 397.689,A -85,B 0,C 180,E1 -523.906,E2 -523.906} C_VEL
LIN {X 0,Y 608.48,Z 397.828,A -85,B 0,C 180,E1 -525.98,E2 -525.98} C_VEL
LIN {X 0,Y 608.445,Z 402.911,A -85,B 0,C 180,E1 -527.057,E2 -527.057} C_VEL
LIN {X 0,Y 608.557,Z 507.78,A -85,B 0,C 180,E1 -528.319,E2 -528.319} C_VEL
LIN {X 0,Y 608.526,Z 521.122,A -85,B 0,C 180,E1 -528.614,E2 -528.614} C_VEL
LIN {X 0,Y 608.523,Z 534.424,A -85,B 0,C 180,E1 -529.057,E2 -529.057} C_VEL
LIN {X 0,Y 608.499,Z 546.37,A -85,B 0,C 180,E1 -529.603,E2 -529.603} C_VEL
LIN {X 0,Y 608.504,Z 557.791,A -85,B 0,C 180,E1 -530.275,E2 -530.275} C_VEL
LIN {X 0,Y 608.474,Z 568.085,A -85,B 0,C 180,E1 -531.029,E2 -531.029} C_VEL
LIN {X 0,Y 608.464,Z 577.35,A -85,B 0,C 180,E1 -531.866,E2 -531.866} C_VEL
LIN {X 0,Y 608.466,Z 586.324,A -85,B 0,C 180,E1 -532.867,E2 -532.867} C_VEL
LIN {X 0,Y 608.444,Z 593.556,A -85,B 0,C 180,E1 -533.867,E2 -533.867} C_VEL
LIN {X 0,Y 608.462,Z 598.435,A -85,B 0,C 180,E1 -534.698,E2 -534.698} C_VEL
LIN {X 0,Y 608.439,Z 603.178,A -85,B 0,C 180,E1 -535.694,E2 -535.694} C_VEL
LIN {X 0,Y 608.425,Z 606.812,A -85,B 0,C 180,E1 -536.689,E2 -536.689} C_VEL
LIN {X 0,Y 608.425,Z 608.691,A -85,B 0,C 180,E1 -537.352,E2 -537.352} C_VEL
LIN {X 0,Y 608.444,Z 610.127,A -85,B 0,C 180,E1 -538.014,E2 -538.014} C_VEL
LIN {X 0,Y 608.439,Z 611.752,A -85,B 0,C 180,E1 -539.338,E2 -539.338} C_VEL
LIN {X 0,Y 608.435,Z 611.995,A -85,B 0,C 180,E1 -540,E2 -540} C_VEL
LIN {X 0,Y 608.438,Z 611.815,A -85,B 0,C 180,E1 -540.662,E2 -540.662} C_VEL
LIN {X 0,Y 608.444,Z 610.276,A -85,B 0,C 180,E1 -541.986,E2 -541.986} C_VEL
LIN {X 0,Y 608.426,Z 608.918,A -85,B 0,C 180,E1 -542.648,E2 -542.648} C_VEL
LIN {X 0,Y 608.449,Z 606.041,A -85,B 0,C 180,E1 -543.642,E2 -543.642} C_VEL
LIN {X 0,Y 608.433,Z 602.143,A -85,B 0,C 180,E1 -544.638,E2 -544.638} C_VEL
LIN {X 0,Y 608.449,Z 597.112,A -85,B 0,C 180,E1 -545.634,E2 -545.634} C_VEL
LIN {X 0,Y 608.441,Z 590.793,A -85,B 0,C 180,E1 -546.633,E2 -546.633} C_VEL
LIN {X 0,Y 608.475,Z 582.877,A -85,B 0,C 180,E1 -547.633,E2 -547.633} C_VEL
LIN {X 0,Y 608.472,Z 573.036,A -85,B 0,C 180,E1 -548.636,E2 -548.636} C_VEL
LIN {X 0,Y 608.477,Z 570.935,A -85,B 0,C 180,E1 -548.819,E2 -548.819} C_VEL
LIN {X 0,Y 607.804,Z 566.604,A -85,B 0,C 180,E1 -549.19,E2 -549.19} C_VEL
LIN {X 0,Y 604.943,Z 559.356,A -85,B 0,C 180,E1 -549.769,E2 -549.769} C_VEL
LIN {X 0,Y 602.126,Z 551.7,A -85,B 0,C 180,E1 -550.302,E2 -550.302} C_VEL
LIN {X 0,Y 601.524,Z 546.644,A -85,B 0,C 180,E1 -550.595,E2 -550.595} C_VEL
LIN {X 0,Y 601.544,Z 534.765,A -85,B 0,C 180,E1 -551.147,E2 -551.147} C_VEL
LIN {X 0,Y 601.583,Z 522.072,A -85,B 0,C 180,E1 -551.583,E2 -551.583} C_VEL
LIN {X 0,Y 601.613,Z 508.053,A -85,B 0,C 180,E1 -551.903,E2 -551.903} C_VEL
LIN {X 0,Y 601.519,Z 403.881,A -85,B 0,C 180,E1 -553.17,E2 -553.17} C_VEL
LIN {X 0,Y 601.386,Z 402.882,A -85,B 0,C 180,E1 -553.194,E2 -553.194} C_VEL
LIN {X 0,Y 601.401,Z 398.569,A -85,B 0,C 180,E1 -554.148,E2 -554.148} C_VEL
LIN {X 0,Y 601.403,Z 398.568,A -85,B 0,C 180,E1 -556.987,E2 -556.987} C_VEL
LIN {X 0,Y 601.4,Z 398.572,A -85,B 0,C 180,E1 -559.81,E2 -559.81} C_VEL
LIN {X 0,Y 601.404,Z 398.566,A -85,B 0,C 180,E1 -562.683,E2 -562.683} C_VEL
LIN {X 0,Y 601.393,Z 398.57,A -85,B 0,C 180,E1 -564.879,E2 -564.879} C_VEL
LIN {X 0,Y 601.415,Z 398.573,A -85,B 0,C 180,E1 -567.362,E2 -567.362} C_VEL
LIN {X 0,Y 601.432,Z 398.562,A -85,B 0,C 180,E1 -570.164,E2 -570.164} C_VEL
LIN {X 0,Y 601.415,Z 398.568,A -85,B 0,C 180,E1 -572.714,E2 -572.714} C_VEL
LIN {X 0,Y 601.392,Z 398.577,A -85,B 0,C 180,E1 -575.111,E2 -575.111} C_VEL
LIN {X 0,Y 601.438,Z 398.565,A -85,B 0,C 180,E1 -577.419,E2 -577.419} C_VEL
LIN {X 0,Y 601.405,Z 398.565,A -85,B 0,C 180,E1 -579.996,E2 -579.996} C_VEL
LIN {X 0,Y 601.412,Z 398.572,A -85,B 0,C 180,E1 -582.67,E2 -582.67} C_VEL
LIN {X 0,Y 601.402,Z 398.566,A -85,B 0,C 180,E1 -585.479,E2 -585.479} C_VEL
LIN {X 0,Y 601.408,Z 398.566,A -85,B 0,C 180,E1 -587.41,E2 -587.41} C_VEL
LIN {X 0,Y 601.404,Z 398.567,A -85,B 0,C 180,E1 -590.004,E2 -590.004} C_VEL
LIN {X 0,Y 601.435,Z 398.572,A -85,B 0,C 180,E1 -592.618,E2 -592.618} C_VEL
LIN {X 0,Y 601.388,Z 398.57,A -85,B 0,C 180,E1 -595.066,E2 -595.066} C_VEL
LIN {X 0,Y 601.407,Z 398.565,A -85,B 0,C 180,E1 -597.483,E2 -597.483} C_VEL
LIN {X 0,Y 601.41,Z 398.567,A -85,B 0,C 180,E1 -599.855,E2 -599.855} C_VEL
LIN {X 0,Y 601.384,Z 398.574,A -85,B 0,C 180,E1 -602.644,E2 -602.644} C_VEL
LIN {X 0,Y 601.376,Z 398.57,A -85,B 0,C 180,E1 -605.12,E2 -605.12} C_VEL
LIN {X 0,Y 601.37,Z 398.581,A -85,B 0,C 180,E1 -607.179,E2 -607.179} C_VEL
LIN {X 0,Y 601.674,Z 404.727,A -85,B 0,C 180,E1 -608.051,E2 -608.051} C_VEL
LIN {X 0,Y 601.596,Z 425.433,A -85,B 0,C 180,E1 -610.907,E2 -610.907} C_VEL
LIN {X 0,Y 601.519,Z 446.139,A -85,B 0,C 180,E1 -613.715,E2 -613.715} C_VEL
LIN {X 0,Y 601.467,Z 466.847,A -85,B 0,C 180,E1 -616.485,E2 -616.485} C_VEL
LIN {X 0,Y 601.47,Z 469.967,A -85,B 0,C 180,E1 -616.872,E2 -616.872} C_VEL
LIN {X 0,Y 601.586,Z 577.754,A -85,B 0,C 180,E1 -618.182,E2 -618.182} C_VEL
LIN {X 0,Y 601.552,Z 590.385,A -85,B 0,C 180,E1 -618.459,E2 -618.459} C_VEL
LIN {X 0,Y 601.534,Z 603.606,A -85,B 0,C 180,E1 -618.896,E2 -618.896} C_VEL
LIN {X 0,Y 601.516,Z 614.75,A -85,B 0,C 180,E1 -619.396,E2 -619.396} C_VEL
LIN {X 0,Y 601.484,Z 626.513,A -85,B 0,C 180,E1 -620.076,E2 -620.076} C_VEL
LIN {X 0,Y 601.444,Z 637.028,A -85,B 0,C 180,E1 -620.839,E2 -620.839} C_VEL
LIN {X 0,Y 601.429,Z 645.638,A -85,B 0,C 180,E1 -621.601,E2 -621.601} C_VEL
LIN {X 0,Y 601.418,Z 653.569,A -85,B 0,C 180,E1 -622.446,E2 -622.446} C_VEL
LIN {X 0,Y 601.377,Z 660.888,A -85,B 0,C 180,E1 -623.393,E2 -623.393} C_VEL
LIN {X 0,Y 601.372,Z 666.612,A -85,B 0,C 180,E1 -624.299,E2 -624.299} C_VEL
LIN {X 0,Y 601.335,Z 671.75,A -85,B 0,C 180,E1 -625.307,E2 -625.307} C_VEL
LIN {X 0,Y 601.367,Z 675.74,A -85,B 0,C 180,E1 -626.315,E2 -626.315} C_VEL
LIN {X 0,Y 601.324,Z 678.694,A -85,B 0,C 180,E1 -627.32,E2 -627.32} C_VEL
LIN {X 0,Y 601.342,Z 680.129,A -85,B 0,C 180,E1 -627.991,E2 -627.991} C_VEL
LIN {X 0,Y 601.339,Z 681.753,A -85,B 0,C 180,E1 -629.33,E2 -629.33} C_VEL
LIN {X 0,Y 601.336,Z 681.996,A -85,B 0,C 180,E1 -630,E2 -630} C_VEL
LIN {X 0,Y 601.339,Z 681.815,A -85,B 0,C 180,E1 -630.67,E2 -630.67} C_VEL
LIN {X 0,Y 601.343,Z 680.277,A -85,B 0,C 180,E1 -632.009,E2 -632.009} C_VEL
LIN {X 0,Y 601.326,Z 678.908,A -85,B 0,C 180,E1 -632.68,E2 -632.68} C_VEL
LIN {X 0,Y 601.368,Z 676.033,A -85,B 0,C 180,E1 -633.685,E2 -633.685} C_VEL
LIN {X 0,Y 601.337,Z 672.133,A -85,B 0,C 180,E1 -634.693,E2 -634.693} C_VEL
LIN {X 0,Y 601.373,Z 667.104,A -85,B 0,C 180,E1 -635.701,E2 -635.701} C_VEL
LIN {X 0,Y 601.382,Z 660.79,A -85,B 0,C 180,E1 -636.711,E2 -636.711} C_VEL
LIN {X 0,Y 601.396,Z 652.874,A -85,B 0,C 180,E1 -637.723,E2 -637.723} C_VEL
LIN {X 0,Y 601.422,Z 644.807,A -85,B 0,C 180,E1 -638.569,E2 -638.569} C_VEL
LIN {X 0,Y 601.453,Z 634.964,A -85,B 0,C 180,E1 -639.415,E2 -639.415} C_VEL
LIN {X 0,Y 601.499,Z 623.919,A -85,B 0,C 180,E1 -640.179,E2 -640.179} C_VEL
LIN {X 0,Y 601.522,Z 611.528,A -85,B 0,C 180,E1 -640.851,E2 -640.851} C_VEL
LIN {X 0,Y 601.552,Z 599.395,A -85,B 0,C 180,E1 -641.35,E2 -641.35} C_VEL
LIN {X 0,Y 601.551,Z 587.265,A -85,B 0,C 180,E1 -641.712,E2 -641.712} C_VEL
LIN {X 0,Y 601.59,Z 573.755,A -85,B 0,C 180,E1 -641.968,E2 -641.968} C_VEL
LIN {X 0,Y 601.484,Z 470.305,A -85,B 0,C 180,E1 -643.213,E2 -643.213} C_VEL
LIN {X 0,Y 601.455,Z 469.466,A -85,B 0,C 180,E1 -643.257,E2 -643.257} C_VEL
LIN {X 0,Y 601.519,Z 448.102,A -85,B 0,C 180,E1 -646.11,E2 -646.11} C_VEL
LIN {X 0,Y 601.598,Z 426.091,A -85,B 0,C 180,E1 -649.093,E2 -649.093} C_VEL
LIN {X 0,Y 601.668,Z 405.373,A -85,B 0,C 180,E1 -651.949,E2 -651.949} C_VEL
LIN {X 0,Y 601.431,Z 398.899,A -85,B 0,C 180,E1 -652.864,E2 -652.864} C_VEL
LIN {X 0,Y 601.392,Z 398.572,A -85,B 0,C 180,E1 -652.956,E2 -652.956} C_VEL
LIN {X 0,Y 601.409,Z 398.574,A -85,B 0,C 180,E1 -655.619,E2 -655.619} C_VEL
LIN {X 0,Y 601.399,Z 398.567,A -85,B 0,C 180,E1 -658.629,E2 -658.629} C_VEL
LIN {X 0,Y 601.418,Z 398.573,A -85,B 0,C 180,E1 -661.454,E2 -661.454} C_VEL
LIN {X 0,Y 601.426,Z 398.565,A -85,B 0,C 180,E1 -664.119,E2 -664.119} C_VEL
LIN {X 0,Y 601.393,Z 398.568,A -85,B 0,C 180,E1 -666.584,E2 -666.584} C_VEL
LIN {X 0,Y 601.406,Z 398.574,A -85,B 0,C 180,E1 -669.127,E2 -669.127} C_VEL
LIN {X 0,Y 601.426,Z 398.565,A -85,B 0,C 180,E1 -671.765,E2 -671.765} C_VEL
LIN {X 0,Y 601.429,Z 398.565,A -85,B 0,C 180,E1 -674.535,E2 -674.535} C_VEL
LIN {X 0,Y 601.411,Z 398.568,A -85,B 0,C 180,E1 -677.41,E2 -677.41} C_VEL
LIN {X 0,Y 601.442,Z 398.565,A -85,B 0,C 180,E1 -680.464,E2 -680.464} C_VEL
LIN {X 0,Y 601.397,Z 398.567,A -85,B 0,C 180,E1 -683.416,E2 -683.416} C_VEL
LIN {X 0,Y 601.433,Z 398.564,A -85,B 0,C 180,E1 -686.065,E2 -686.065} C_VEL
LIN {X 0,Y 601.399,Z 398.569,A -85,B 0,C 180,E1 -689.057,E2 -689.057} C_VEL
LIN {X 0,Y 601.403,Z 398.566,A -85,B 0,C 180,E1 -691.371,E2 -691.371} C_VEL
LIN {X 0,Y 601.411,Z 398.572,A -85,B 0,C 180,E1 -694.134,E2 -694.134} C_VEL
LIN {X 0,Y 601.38,Z 398.576,A -85,B 0,C 180,E1 -696.588,E2 -696.588} C_VEL
LIN {X 0,Y 601.37,Z 398.581,A -85,B 0,C 180,E1 -697.179,E2 -697.179} C_VEL
LIN {X 0,Y 601.674,Z 404.727,A -85,B 0,C 180,E1 -698.051,E2 -698.051} C_VEL
LIN {X 0,Y 601.596,Z 425.433,A -85,B 0,C 180,E1 -700.907,E2 -700.907} C_VEL
LIN {X 0,Y 601.519,Z 446.139,A -85,B 0,C 180,E1 -703.715,E2 -703.715} C_VEL
LIN {X 0,Y 601.467,Z 466.847,A -85,B 0,C 180,E1 -706.485,E2 -706.485} C_VEL
LIN {X 0,Y 601.47,Z 469.965,A -85,B 0,C 180,E1 -706.872,E2 -706.872} C_VEL
LIN {X 0,Y 601.586,Z 577.767,A -85,B 0,C 180,E1 -708.182,E2 -708.182} C_VEL
LIN {X 0,Y 601.56,Z 591.147,A -85,B 0,C 180,E1 -708.48,E2 -708.48} C_VEL
LIN {X 0,Y 601.553,Z 604.392,A -85,B 0,C 180,E1 -708.927,E2 -708.927} C_VEL
LIN {X 0,Y 601.505,Z 616.379,A -85,B 0,C 180,E1 -709.481,E2 -709.481} C_VEL
LIN {X 0,Y 601.472,Z 627.802,A -85,B 0,C 180,E1 -710.16,E2 -710.16} C_VEL
LIN {X 0,Y 601.438,Z 638.095,A -85,B 0,C 180,E1 -710.924,E2 -710.924} C_VEL
LIN {X 0,Y 601.412,Z 647.346,A -85,B 0,C 180,E1 -711.77,E2 -711.77} C_VEL
LIN {X 0,Y 601.388,Z 656.325,A -85,B 0,C 180,E1 -712.783,E2 -712.783} C_VEL
LIN {X 0,Y 601.376,Z 663.468,A -85,B 0,C 180,E1 -713.78,E2 -713.78} C_VEL
LIN {X 0,Y 601.372,Z 668.439,A -85,B 0,C 180,E1 -714.635,E2 -714.635} C_VEL
LIN {X 0,Y 601.354,Z 673.183,A -85,B 0,C 180,E1 -715.643,E2 -715.643} C_VEL
LIN {X 0,Y 601.344,Z 676.817,A -85,B 0,C 180,E1 -716.65,E2 -716.65} C_VEL
LIN {X 0,Y 601.324,Z 678.688,A -85,B 0,C 180,E1 -717.32,E2 -717.32} C_VEL
LIN {X 0,Y 601.342,Z 680.122,A -85,B 0,C 180,E1 -717.991,E2 -717.991} C_VEL
LIN {X 0,Y 601.339,Z 681.752,A -85,B 0,C 180,E1 -719.33,E2 -719.33} C_VEL
LIN {X 0,Y 601.336,Z 681.991,A -85,B 0,C 180,E1 -720,E2 -720} C_VEL
LIN {X 0,Y 601.339,Z 681.814,A -85,B 0,C 180,E1 -720.67,E2 -720.67} C_VEL
LIN {X 0,Y 601.343,Z 680.273,A -85,B 0,C 180,E1 -722.009,E2 -722.009} C_VEL
LIN {X 0,Y 601.326,Z 678.917,A -85,B 0,C 180,E1 -722.68,E2 -722.68} C_VEL
LIN {X 0,Y 601.368,Z 676.043,A -85,B 0,C 180,E1 -723.685,E2 -723.685} C_VEL
LIN {X 0,Y 601.337,Z 672.143,A -85,B 0,C 180,E1 -724.693,E2 -724.693} C_VEL
LIN {X 0,Y 601.373,Z 667.111,A -85,B 0,C 180,E1 -725.701,E2 -725.701} C_VEL
LIN {X 0,Y 601.382,Z 660.778,A -85,B 0,C 180,E1 -726.711,E2 -726.711} C_VEL
LIN {X 0,Y 601.396,Z 652.877,A -85,B 0,C 180,E1 -727.723,E2 -727.723} C_VEL
LIN {X 0,Y 601.436,Z 643.03,A -85,B 0,C 180,E1 -728.738,E2 -728.738} C_VEL
LIN {X 0,Y 601.449,Z 632.695,A -85,B 0,C 180,E1 -729.585,E2 -729.585} C_VEL
LIN {X 0,Y 601.477,Z 622.498,A -85,B 0,C 180,E1 -730.264,E2 -730.264} C_VEL
LIN {X 0,Y 601.531,Z 611.523,A -85,B 0,C 180,E1 -730.851,E2 -730.851} C_VEL
LIN {X 0,Y 601.544,Z 599.734,A -85,B 0,C 180,E1 -731.34,E2 -731.34} C_VEL
LIN {X 0,Y 601.551,Z 587.257,A -85,B 0,C 180,E1 -731.712,E2 -731.712} C_VEL
LIN {X 0,Y 601.59,Z 573.757,A -85,B 0,C 180,E1 -731.968,E2 -731.968} C_VEL
LIN {X 0,Y 601.484,Z 470.308,A -85,B 0,C 180,E1 -733.213,E2 -733.213} C_VEL
LIN {X 0,Y 601.455,Z 469.466,A -85,B 0,C 180,E1 -733.257,E2 -733.257} C_VEL
LIN {X 0,Y 601.519,Z 448.103,A -85,B 0,C 180,E1 -736.11,E2 -736.11} C_VEL
LIN {X 0,Y 601.598,Z 426.091,A -85,B 0,C 180,E1 -739.093,E2 -739.093} C_VEL
LIN {X 0,Y 601.668,Z 405.374,A -85,B 0,C 180,E1 -741.949,E2 -741.949} C_VEL
LIN {X 0,Y 601.431,Z 398.899,A -85,B 0,C 180,E1 -742.864,E2 -742.864} C_VEL
LIN {X 0,Y 601.392,Z 398.572,A -85,B 0,C 180,E1 -742.956,E2 -742.956} C_VEL
LIN {X 0,Y 601.409,Z 398.574,A -85,B 0,C 180,E1 -745.619,E2 -745.619} C_VEL
LIN {X 0,Y 601.4,Z 398.567,A -85,B 0,C 180,E1 -748.629,E2 -748.629} C_VEL
LIN {X 0,Y 601.417,Z 398.574,A -85,B 0,C 180,E1 -751.454,E2 -751.454} C_VEL
LIN {X 0,Y 601.426,Z 398.564,A -85,B 0,C 180,E1 -754.119,E2 -754.119} C_VEL
LIN {X 0,Y 601.394,Z 398.568,A -85,B 0,C 180,E1 -756.584,E2 -756.584} C_VEL
LIN {X 0,Y 601.407,Z 398.574,A -85,B 0,C 180,E1 -759.127,E2 -759.127} C_VEL
LIN {X 0,Y 601.427,Z 398.565,A -85,B 0,C 180,E1 -761.765,E2 -761.765} C_VEL
LIN {X 0,Y 601.428,Z 398.566,A -85,B 0,C 180,E1 -764.535,E2 -764.535} C_VEL
LIN {X 0,Y 601.411,Z 398.568,A -85,B 0,C 180,E1 -767.41,E2 -767.41} C_VEL
LIN {X 0,Y 601.405,Z 398.566,A -85,B 0,C 180,E1 -770.004,E2 -770.004} C_VEL
LIN {X 0,Y 601.437,Z 398.57,A -85,B 0,C 180,E1 -772.618,E2 -772.618} C_VEL
LIN {X 0,Y 601.393,Z 398.571,A -85,B 0,C 180,E1 -775.066,E2 -775.066} C_VEL
LIN {X 0,Y 601.41,Z 398.565,A -85,B 0,C 180,E1 -777.483,E2 -777.483} C_VEL
LIN {X 0,Y 601.409,Z 398.567,A -85,B 0,C 180,E1 -779.855,E2 -779.855} C_VEL
LIN {X 0,Y 601.384,Z 398.574,A -85,B 0,C 180,E1 -782.644,E2 -782.644} C_VEL
LIN {X 0,Y 601.407,Z 398.724,A -85,B 0,C 180,E1 -785.029,E2 -785.029} C_VEL
LIN {X 0,Y 601.832,Z 403.441,A -85,B 0,C 180,E1 -785.625,E2 -785.625} C_VEL
LIN {X 0,Y 601.681,Z 426.573,A -85,B 0,C 180,E1 -788.411,E2 -788.411} C_VEL
LIN {X 0,Y 601.634,Z 447.647,A -85,B 0,C 180,E1 -790.908,E2 -790.908} C_VEL
LIN {X 0,Y 601.537,Z 471.732,A -85,B 0,C 180,E1 -793.716,E2 -793.716} C_VEL
LIN {X 0,Y 601.445,Z 495.817,A -85,B 0,C 180,E1 -796.485,E2 -796.485} C_VEL
LIN {X 0,Y 601.427,Z 498.64,A -85,B 0,C 180,E1 -796.807,E2 -796.807} C_VEL
LIN {X 0,Y 601.654,Z 528.756,A -85,B 0,C 180,E1 -797.177,E2 -797.177} C_VEL
LIN {X 0,Y 601.603,Z 607.943,A -85,B 0,C 180,E1 -798.139,E2 -798.139} C_VEL
LIN {X 0,Y 601.563,Z 621.215,A -85,B 0,C 180,E1 -798.438,E2 -798.438} C_VEL
LIN {X 0,Y 601.543,Z 632.911,A -85,B 0,C 180,E1 -798.826,E2 -798.826} C_VEL
LIN {X 0,Y 601.516,Z 645.633,A -85,B 0,C 180,E1 -799.396,E2 -799.396} C_VEL
LIN {X 0,Y 601.484,Z 657.198,A -85,B 0,C 180,E1 -800.076,E2 -800.076} C_VEL
LIN {X 0,Y 601.444,Z 667.594,A -85,B 0,C 180,E1 -800.839,E2 -800.839} C_VEL
LIN {X 0,Y 601.429,Z 676.111,A -85,B 0,C 180,E1 -801.601,E2 -801.601} C_VEL
LIN {X 0,Y 601.418,Z 683.96,A -85,B 0,C 180,E1 -802.446,E2 -802.446} C_VEL
LIN {X 0,Y 601.37,Z 691.224,A -85,B 0,C 180,E1 -803.398,E2 -803.398} C_VEL
LIN {X 0,Y 601.372,Z 696.866,A -85,B 0,C 180,E1 -804.299,E2 -804.299} C_VEL
LIN {X 0,Y 601.336,Z 701.95,A -85,B 0,C 180,E1 -805.307,E2 -805.307} C_VEL
LIN {X 0,Y 601.368,Z 705.896,A -85,B 0,C 180,E1 -806.315,E2 -806.315} C_VEL
LIN {X 0,Y 601.325,Z 708.809,A -85,B 0,C 180,E1 -807.32,E2 -807.32} C_VEL
LIN {X 0,Y 601.343,Z 710.202,A -85,B 0,C 180,E1 -807.991,E2 -807.991} C_VEL
LIN {X 0,Y 601.339,Z 711.784,A -85,B 0,C 180,E1 -809.33,E2 -809.33} C_VEL
LIN {X 0,Y 601.335,Z 712,A -85,B 0,C 180,E1 -810,E2 -810} C_VEL
LIN {X 0,Y 601.347,Z 711.184,A -85,B 0,C 180,E1 -811.339,E2 -811.339} C_VEL
LIN {X 0,Y 601.343,Z 710.202,A -85,B 0,C 180,E1 -812.009,E2 -812.009} C_VEL
LIN {X 0,Y 601.325,Z 708.809,A -85,B 0,C 180,E1 -812.68,E2 -812.68} C_VEL
LIN {X 0,Y 601.368,Z 705.896,A -85,B 0,C 180,E1 -813.685,E2 -813.685} C_VEL
LIN {X 0,Y 601.336,Z 701.95,A -85,B 0,C 180,E1 -814.693,E2 -814.693} C_VEL
LIN {X 0,Y 601.372,Z 695.877,A -85,B 0,C 180,E1 -815.869,E2 -815.869} C_VEL
LIN {X 0,Y 601.382,Z 689.235,A -85,B 0,C 180,E1 -816.88,E2 -816.88} C_VEL
LIN {X 0,Y 601.401,Z 680.989,A -85,B 0,C 180,E1 -817.892,E2 -817.892} C_VEL
LIN {X 0,Y 601.436,Z 672.536,A -85,B 0,C 180,E1 -818.738,E2 -818.738} C_VEL
LIN {X 0,Y 601.448,Z 662.091,A -85,B 0,C 180,E1 -819.585,E2 -819.585} C_VEL
LIN {X 0,Y 601.478,Z 651.756,A -85,B 0,C 180,E1 -820.264,E2 -820.264} C_VEL
LIN {X 0,Y 601.535,Z 640.91,A -85,B 0,C 180,E1 -820.835,E2 -820.835} C_VEL
LIN {X 0,Y 601.544,Z 628.381,A -85,B 0,C 180,E1 -821.341,E2 -821.341} C_VEL
LIN {X 0,Y 601.554,Z 615.349,A -85,B 0,C 180,E1 -821.712,E2 -821.712} C_VEL
LIN {X 0,Y 601.61,Z 602.079,A -85,B 0,C 180,E1 -821.946,E2 -821.946} C_VEL
LIN {X 0,Y 601.528,Z 499.243,A -85,B 0,C 180,E1 -823.18,E2 -823.18} C_VEL
LIN {X 0,Y 601.423,Z 498.452,A -85,B 0,C 180,E1 -823.215,E2 -823.215} C_VEL
LIN {X 0,Y 601.554,Z 474.743,A -85,B 0,C 180,E1 -825.935,E2 -825.935} C_VEL
LIN {X 0,Y 601.631,Z 450.513,A -85,B 0,C 180,E1 -828.755,E2 -828.755} C_VEL
LIN {X 0,Y 601.679,Z 428.078,A -85,B 0,C 180,E1 -831.409,E2 -831.409} C_VEL
LIN {X 0,Y 601.806,Z 405.498,A -85,B 0,C 180,E1 -834.126,E2 -834.126} C_VEL
LIN {X 0,Y 601.532,Z 399.477,A -85,B 0,C 180,E1 -834.873,E2 -834.873} C_VEL
LIN {X 0,Y 601.382,Z 398.574,A -85,B 0,C 180,E1 -835.018,E2 -835.018} C_VEL
LIN {X 0,Y 601.389,Z 398.576,A -85,B 0,C 180,E1 -837.869,E2 -837.869} C_VEL
LIN {X 0,Y 601.407,Z 398.568,A -85,B 0,C 180,E1 -840.165,E2 -840.165} C_VEL
LIN {X 0,Y 601.4,Z 398.567,A -85,B 0,C 180,E1 -842.712,E2 -842.712} C_VEL
LIN {X 0,Y 601.378,Z 398.573,A -85,B 0,C 180,E1 -845.109,E2 -845.109} C_VEL
LIN {X 0,Y 601.434,Z 398.572,A -85,B 0,C 180,E1 -847.419,E2 -847.419} C_VEL
LIN {X 0,Y 601.403,Z 398.568,A -85,B 0,C 180,E1 -849.996,E2 -849.996} C_VEL
LIN {X 0,Y 601.387,Z 398.569,A -85,B 0,C 180,E1 -852.673,E2 -852.673} C_VEL
LIN {X 0,Y 601.43,Z 398.569,A -85,B 0,C 180,E1 -855.482,E2 -855.482} C_VEL
LIN {X 0,Y 601.421,Z 398.564,A -85,B 0,C 180,E1 -858.408,E2 -858.408} C_VEL
LIN {X 0,Y 601.436,Z 398.565,A -85,B 0,C 180,E1 -861.529,E2 -861.529} C_VEL
LIN {X 0,Y 601.389,Z 398.568,A -85,B 0,C 180,E1 -864.245,E2 -864.245} C_VEL
LIN {X 0,Y 601.417,Z 398.57,A -85,B 0,C 180,E1 -866.686,E2 -866.686} C_VEL
LIN {X 0,Y 601.416,Z 398.572,A -85,B 0,C 180,E1 -869.058,E2 -869.058} C_VEL
LIN {X 0,Y 601.419,Z 398.566,A -85,B 0,C 180,E1 -871.372,E2 -871.372} C_VEL
LIN {X 0,Y 601.396,Z 398.567,A -85,B 0,C 180,E1 -873.636,E2 -873.636} C_VEL
LIN {X 0,Y 601.418,Z 398.573,A -85,B 0,C 180,E1 -876.59,E2 -876.59} C_VEL
LIN {X 0,Y 601.415,Z 398.565,A -85,B 0,C 180,E1 -879.478,E2 -879.478} C_VEL
LIN {X 0,Y 601.394,Z 398.574,A -85,B 0,C 180,E1 -882.312,E2 -882.312} C_VEL
LIN {X 0,Y 601.406,Z 398.575,A -85,B 0,C 180,E1 -884.408,E2 -884.408} C_VEL
LIN {X 0,Y 601.436,Z 398.656,A -85,B 0,C 180,E1 -885.99,E2 -885.99} C_VEL
LIN {X 0,Y 601.388,Z 402.864,A -85,B 0,C 180,E1 -886.892,E2 -886.892} C_VEL
LIN {X 0,Y 601.665,Z 407.123,A -85,B 0,C 180,E1 -886.963,E2 -886.963} C_VEL
LIN {X 0,Y 601.603,Z 507.772,A -85,B 0,C 180,E1 -888.182,E2 -888.182} C_VEL
LIN {X 0,Y 601.59,Z 521.151,A -85,B 0,C 180,E1 -888.481,E2 -888.481} C_VEL
LIN {X 0,Y 601.537,Z 533.573,A -85,B 0,C 180,E1 -888.895,E2 -888.895} C_VEL
LIN {X 0,Y 601.517,Z 544.727,A -85,B 0,C 180,E1 -889.396,E2 -889.396} C_VEL
LIN {X 0,Y 601.483,Z 556.526,A -85,B 0,C 180,E1 -890.076,E2 -890.076} C_VEL
LIN {X 0,Y 601.438,Z 568.094,A -85,B 0,C 180,E1 -890.924,E2 -890.924} C_VEL
LIN {X 0,Y 601.411,Z 577.354,A -85,B 0,C 180,E1 -891.77,E2 -891.77} C_VEL
LIN {X 0,Y 601.388,Z 586.331,A -85,B 0,C 180,E1 -892.783,E2 -892.783} C_VEL
LIN {X 0,Y 601.376,Z 593.472,A -85,B 0,C 180,E1 -893.781,E2 -893.781} C_VEL
LIN {X 0,Y 601.372,Z 598.44,A -85,B 0,C 180,E1 -894.635,E2 -894.635} C_VEL
LIN {X 0,Y 601.354,Z 603.181,A -85,B 0,C 180,E1 -895.643,E2 -895.643} C_VEL
LIN {X 0,Y 601.344,Z 606.811,A -85,B 0,C 180,E1 -896.65,E2 -896.65} C_VEL
LIN {X 0,Y 601.324,Z 608.695,A -85,B 0,C 180,E1 -897.32,E2 -897.32} C_VEL
LIN {X 0,Y 601.343,Z 610.13,A -85,B 0,C 180,E1 -897.991,E2 -897.991} C_VEL
LIN {X 0,Y 601.339,Z 611.754,A -85,B 0,C 180,E1 -899.33,E2 -899.33} C_VEL
LIN {X 0,Y 601.336,Z 611.996,A -85,B 0,C 180,E1 -900,E2 -900} C_VEL
LIN {X 0,Y 601.339,Z 611.816,A -85,B 0,C 180,E1 -900.67,E2 -900.67} C_VEL
LIN {X 0,Y 601.343,Z 610.277,A -85,B 0,C 180,E1 -902.009,E2 -902.009} C_VEL
LIN {X 0,Y 601.326,Z 608.912,A -85,B 0,C 180,E1 -902.68,E2 -902.68} C_VEL
LIN {X 0,Y 601.368,Z 606.037,A -85,B 0,C 180,E1 -903.685,E2 -903.685} C_VEL
LIN {X 0,Y 601.337,Z 602.141,A -85,B 0,C 180,E1 -904.693,E2 -904.693} C_VEL
LIN {X 0,Y 601.373,Z 597.112,A -85,B 0,C 180,E1 -905.701,E2 -905.701} C_VEL
LIN {X 0,Y 601.382,Z 590.784,A -85,B 0,C 180,E1 -906.711,E2 -906.711} C_VEL
LIN {X 0,Y 601.396,Z 582.872,A -85,B 0,C 180,E1 -907.723,E2 -907.723} C_VEL
LIN {X 0,Y 601.437,Z 573.031,A -85,B 0,C 180,E1 -908.738,E2 -908.738} C_VEL
LIN {X 0,Y 601.449,Z 562.696,A -85,B 0,C 180,E1 -909.585,E2 -909.585} C_VEL
LIN {X 0,Y 601.477,Z 552.487,A -85,B 0,C 180,E1 -910.264,E2 -910.264} C_VEL
LIN {X 0,Y 601.524,Z 546.644,A -85,B 0,C 180,E1 -910.595,E2 -910.595} C_VEL
LIN {X 0,Y 600.914,Z 541.514,A -85,B 0,C 180,E1 -910.87,E2 -910.87} C_VEL
LIN {X 0,Y 598.08,Z 533.083,A -85,B 0,C 180,E1 -911.295,E2 -911.295} C_VEL
LIN {X 0,Y 595.246,Z 524.341,A -85,B 0,C 180,E1 -911.65,E2 -911.65} C_VEL
LIN {X 0,Y 594.627,Z 518.731,A -85,B 0,C 180,E1 -911.814,E2 -911.814} C_VEL
LIN {X 0,Y 594.691,Z 506.627,A -85,B 0,C 180,E1 -912.066,E2 -912.066} C_VEL
LIN {X 0,Y 594.665,Z 404.955,A -85,B 0,C 180,E1 -913.311,E2 -913.311} C_VEL
LIN {X 0,Y 594.324,Z 402.88,A -85,B 0,C 180,E1 -913.354,E2 -913.354} C_VEL
LIN {X 0,Y 594.366,Z 399.447,A -85,B 0,C 180,E1 -914.107,E2 -914.107} C_VEL
LIN {X 0,Y 594.373,Z 399.446,A -85,B 0,C 180,E1 -917.194,E2 -917.194} C_VEL
LIN {X 0,Y 594.366,Z 399.445,A -85,B 0,C 180,E1 -920.054,E2 -920.054} C_VEL
LIN {X 0,Y 594.361,Z 399.446,A -85,B 0,C 180,E1 -922.968,E2 -922.968} C_VEL
LIN {X 0,Y 594.371,Z 399.449,A -85,B 0,C 180,E1 -925.193,E2 -925.193} C_VEL
LIN {X 0,Y 594.372,Z 399.448,A -85,B 0,C 180,E1 -927.523,E2 -927.523} C_VEL
LIN {X 0,Y 594.389,Z 399.44,A -85,B 0,C 180,E1 -930.328,E2 -930.328} C_VEL
LIN {X 0,Y 594.378,Z 399.447,A -85,B 0,C 180,E1 -932.95,E2 -932.95} C_VEL
LIN {X 0,Y 594.351,Z 399.449,A -85,B 0,C 180,E1 -935.409,E2 -935.409} C_VEL
LIN {X 0,Y 594.39,Z 399.44,A -85,B 0,C 180,E1 -937.941,E2 -937.941} C_VEL
LIN {X 0,Y 594.379,Z 399.449,A -85,B 0,C 180,E1 -940.822,E2 -940.822} C_VEL
LIN {X 0,Y 594.369,Z 399.446,A -85,B 0,C 180,E1 -943.3,E2 -943.3} C_VEL
LIN {X 0,Y 594.379,Z 399.442,A -85,B 0,C 180,E1 -946.16,E2 -946.16} C_VEL
LIN {X 0,Y 594.374,Z 399.444,A -85,B 0,C 180,E1 -949.179,E2 -949.179} C_VEL
LIN {X 0,Y 594.382,Z 399.443,A -85,B 0,C 180,E1 -952.059,E2 -952.059} C_VEL
LIN {X 0,Y 594.348,Z 399.453,A -85,B 0,C 180,E1 -954.677,E2 -954.677} C_VEL
LIN {X 0,Y 594.376,Z 399.443,A -85,B 0,C 180,E1 -957.089,E2 -957.089} C_VEL
LIN {X 0,Y 594.371,Z 399.443,A -85,B 0,C 180,E1 -959.675,E2 -959.675} C_VEL
LIN {X 0,Y 594.345,Z 399.454,A -85,B 0,C 180,E1 -962.482,E2 -962.482} C_VEL
LIN {X 0,Y 594.335,Z 399.45,A -85,B 0,C 180,E1 -964.805,E2 -964.805} C_VEL
LIN {X 0,Y 594.348,Z 399.556,A -85,B 0,C 180,E1 -967.032,E2 -967.032} C_VEL
LIN {X 0,Y 594.766,Z 404.732,A -85,B 0,C 180,E1 -967.782,E2 -967.782} C_VEL
LIN {X 0,Y 594.646,Z 424.143,A -85,B 0,C 180,E1 -970.495,E2 -970.495} C_VEL
LIN {X 0,Y 594.511,Z 442.993,A -85,B 0,C 180,E1 -973.087,E2 -973.087} C_VEL
LIN {X 0,Y 594.474,Z 464.946,A -85,B 0,C 180,E1 -976.066,E2 -976.066} C_VEL
LIN {X 0,Y 594.455,Z 470.013,A -85,B 0,C 180,E1 -976.715,E2 -976.715} C_VEL
LIN {X 0,Y 594.716,Z 477.165,A -85,B 0,C 180,E1 -976.807,E2 -976.807} C_VEL
LIN {X 0,Y 594.654,Z 577.735,A -85,B 0,C 180,E1 -978.042,E2 -978.042} C_VEL
LIN {X 0,Y 594.603,Z 590.412,A -85,B 0,C 180,E1 -978.322,E2 -978.322} C_VEL
LIN {X 0,Y 594.561,Z 603.083,A -85,B 0,C 180,E1 -978.744,E2 -978.744} C_VEL
LIN {X 0,Y 594.529,Z 614.758,A -85,B 0,C 180,E1 -979.27,E2 -979.27} C_VEL
LIN {X 0,Y 594.461,Z 625.203,A -85,B 0,C 180,E1 -979.871,E2 -979.871} C_VEL
LIN {X 0,Y 594.405,Z 635.974,A -85,B 0,C 180,E1 -980.644,E2 -980.644} C_VEL
LIN {X 0,Y 594.384,Z 645.643,A -85,B 0,C 180,E1 -981.501,E2 -981.501} C_VEL
LIN {X 0,Y 594.337,Z 654.972,A -85,B 0,C 180,E1 -982.526,E2 -982.526} C_VEL
LIN {X 0,Y 594.285,Z 662.85,A -85,B 0,C 180,E1 -983.612,E2 -983.612} C_VEL
LIN {X 0,Y 594.289,Z 668.432,A -85,B 0,C 180,E1 -984.571,E2 -984.571} C_VEL
LIN {X 0,Y 594.27,Z 673.169,A -85,B 0,C 180,E1 -985.591,E2 -985.591} C_VEL
LIN {X 0,Y 594.267,Z 676.807,A -85,B 0,C 180,E1 -986.61,E2 -986.61} C_VEL
LIN {X 0,Y 594.225,Z 678.694,A -85,B 0,C 180,E1 -987.288,E2 -987.288} C_VEL
LIN {X 0,Y 594.241,Z 680.131,A -85,B 0,C 180,E1 -987.967,E2 -987.967} C_VEL
LIN {X 0,Y 594.24,Z 681.754,A -85,B 0,C 180,E1 -989.322,E2 -989.322} C_VEL
LIN {X 0,Y 594.236,Z 681.996,A -85,B 0,C 180,E1 -990,E2 -990} C_VEL
LIN {X 0,Y 594.239,Z 681.814,A -85,B 0,C 180,E1 -990.678,E2 -990.678} C_VEL
LIN {X 0,Y 594.242,Z 680.277,A -85,B 0,C 180,E1 -992.033,E2 -992.033} C_VEL
LIN {X 0,Y 594.226,Z 678.899,A -85,B 0,C 180,E1 -992.712,E2 -992.712} C_VEL
LIN {X 0,Y 594.289,Z 676.024,A -85,B 0,C 180,E1 -993.729,E2 -993.729} C_VEL
LIN {X 0,Y 594.241,Z 672.125,A -85,B 0,C 180,E1 -994.749,E2 -994.749} C_VEL
LIN {X 0,Y 594.299,Z 667.098,A -85,B 0,C 180,E1 -995.769,E2 -995.769} C_VEL
LIN {X 0,Y 594.316,Z 660.786,A -85,B 0,C 180,E1 -996.791,E2 -996.791} C_VEL
LIN {X 0,Y 594.347,Z 652.87,A -85,B 0,C 180,E1 -997.816,E2 -997.816} C_VEL
LIN {X 0,Y 594.366,Z 644.801,A -85,B 0,C 180,E1 -998.671,E2 -998.671} C_VEL
LIN {X 0,Y 594.415,Z 634.944,A -85,B 0,C 180,E1 -999.528,E2 -999.528} C_VEL
LIN {X 0,Y 594.471,Z 623.914,A -85,B 0,C 180,E1 -1000.301,E2 -1000.301} C_VEL
LIN {X 0,Y 594.551,Z 611.505,A -85,B 0,C 180,E1 -1000.981,E2 -1000.981} C_VEL
LIN {X 0,Y 594.579,Z 599.594,A -85,B 0,C 180,E1 -1001.477,E2 -1001.477} C_VEL
LIN {X 0,Y 594.615,Z 587.215,A -85,B 0,C 180,E1 -1001.851,E2 -1001.851} C_VEL
LIN {X 0,Y 594.658,Z 573.716,A -85,B 0,C 180,E1 -1002.109,E2 -1002.109} C_VEL
LIN {X 0,Y 594.565,Z 470.707,A -85,B 0,C 180,E1 -1003.365,E2 -1003.365} C_VEL
LIN {X 0,Y 594.4,Z 469.623,A -85,B 0,C 180,E1 -1003.395,E2 -1003.395} C_VEL
LIN {X 0,Y 594.524,Z 449.393,A -85,B 0,C 180,E1 -1006.129,E2 -1006.129} C_VEL
LIN {X 0,Y 594.631,Z 427.729,A -85,B 0,C 180,E1 -1009.098,E2 -1009.098} C_VEL
LIN {X 0,Y 594.756,Z 406.664,A -85,B 0,C 180,E1 -1012.035,E2 -1012.035} C_VEL
LIN {X 0,Y 594.653,Z 401.282,A -85,B 0,C 180,E1 -1012.801,E2 -1012.801} C_VEL
LIN {X 0,Y 594.349,Z 399.451,A -85,B 0,C 180,E1 -1013.106,E2 -1013.106} C_VEL
LIN {X 0,Y 594.364,Z 399.451,A -85,B 0,C 180,E1 -1015.945,E2 -1015.945} C_VEL
LIN {X 0,Y 594.373,Z 399.443,A -85,B 0,C 180,E1 -1018.999,E2 -1018.999} C_VEL
LIN {X 0,Y 594.375,Z 399.451,A -85,B 0,C 180,E1 -1021.642,E2 -1021.642} C_VEL
LIN {X 0,Y 594.37,Z 399.443,A -85,B 0,C 180,E1 -1024.581,E2 -1024.581} C_VEL
LIN {X 0,Y 594.39,Z 399.445,A -85,B 0,C 180,E1 -1027.608,E2 -1027.608} C_VEL
LIN {X 0,Y 594.367,Z 399.443,A -85,B 0,C 180,E1 -1030.567,E2 -1030.567} C_VEL
LIN {X 0,Y 594.37,Z 399.449,A -85,B 0,C 180,E1 -1033.3,E2 -1033.3} C_VEL
LIN {X 0,Y 594.371,Z 399.443,A -85,B 0,C 180,E1 -1036.161,E2 -1036.161} C_VEL
LIN {X 0,Y 594.383,Z 399.444,A -85,B 0,C 180,E1 -1038.536,E2 -1038.536} C_VEL
LIN {X 0,Y 594.38,Z 399.444,A -85,B 0,C 180,E1 -1041.297,E2 -1041.297} C_VEL
LIN {X 0,Y 594.352,Z 399.443,A -85,B 0,C 180,E1 -1043.755,E2 -1043.755} C_VEL
LIN {X 0,Y 594.379,Z 399.445,A -85,B 0,C 180,E1 -1046.239,E2 -1046.239} C_VEL
LIN {X 0,Y 594.366,Z 399.451,A -85,B 0,C 180,E1 -1048.649,E2 -1048.649} C_VEL
LIN {X 0,Y 594.376,Z 399.443,A -85,B 0,C 180,E1 -1051.044,E2 -1051.044} C_VEL
LIN {X 0,Y 594.37,Z 399.448,A -85,B 0,C 180,E1 -1054.055,E2 -1054.055} C_VEL
LIN {X 0,Y 594.347,Z 399.451,A -85,B 0,C 180,E1 -1056.94,E2 -1056.94} C_VEL
LIN {X 0,Y 594.35,Z 399.556,A -85,B 0,C 180,E1 -1057.032,E2 -1057.032} C_VEL
LIN {X 0,Y 594.766,Z 404.732,A -85,B 0,C 180,E1 -1057.782,E2 -1057.782} C_VEL
LIN {X 0,Y 594.646,Z 424.143,A -85,B 0,C 180,E1 -1060.495,E2 -1060.495} C_VEL
LIN {X 0,Y 594.511,Z 442.992,A -85,B 0,C 180,E1 -1063.087,E2 -1063.087} C_VEL
LIN {X 0,Y 594.475,Z 464.928,A -85,B 0,C 180,E1 -1066.064,E2 -1066.064} C_VEL
LIN {X 0,Y 594.455,Z 470.011,A -85,B 0,C 180,E1 -1066.715,E2 -1066.715} C_VEL
LIN {X 0,Y 594.716,Z 477.163,A -85,B 0,C 180,E1 -1066.807,E2 -1066.807} C_VEL
LIN {X 0,Y 594.654,Z 577.753,A -85,B 0,C 180,E1 -1068.042,E2 -1068.042} C_VEL
LIN {X 0,Y 594.602,Z 590.416,A -85,B 0,C 180,E1 -1068.322,E2 -1068.322} C_VEL
LIN {X 0,Y 594.597,Z 603.543,A -85,B 0,C 180,E1 -1068.762,E2 -1068.762} C_VEL
LIN {X 0,Y 594.529,Z 614.73,A -85,B 0,C 180,E1 -1069.27,E2 -1069.27} C_VEL
LIN {X 0,Y 594.483,Z 626.536,A -85,B 0,C 180,E1 -1069.958,E2 -1069.958} C_VEL
LIN {X 0,Y 594.406,Z 638.103,A -85,B 0,C 180,E1 -1070.815,E2 -1070.815} C_VEL
LIN {X 0,Y 594.373,Z 647.341,A -85,B 0,C 180,E1 -1071.672,E2 -1071.672} C_VEL
LIN {X 0,Y 594.317,Z 656.327,A -85,B 0,C 180,E1 -1072.697,E2 -1072.697} C_VEL
LIN {X 0,Y 594.285,Z 662.854,A -85,B 0,C 180,E1 -1073.612,E2 -1073.612} C_VEL
LIN {X 0,Y 594.289,Z 668.444,A -85,B 0,C 180,E1 -1074.571,E2 -1074.571} C_VEL
LIN {X 0,Y 594.27,Z 673.188,A -85,B 0,C 180,E1 -1075.591,E2 -1075.591} C_VEL
LIN {X 0,Y 594.267,Z 676.821,A -85,B 0,C 180,E1 -1076.61,E2 -1076.61} C_VEL
LIN {X 0,Y 594.225,Z 678.685,A -85,B 0,C 180,E1 -1077.288,E2 -1077.288} C_VEL
LIN {X 0,Y 594.241,Z 680.116,A -85,B 0,C 180,E1 -1077.967,E2 -1077.967} C_VEL
LIN {X 0,Y 594.247,Z 681.135,A -85,B 0,C 180,E1 -1078.645,E2 -1078.645} C_VEL
LIN {X 0,Y 594.236,Z 681.983,A -85,B 0,C 180,E1 -1080,E2 -1080} C_VEL
LIN {X 0,Y 594.239,Z 681.813,A -85,B 0,C 180,E1 -1080.678,E2 -1080.678} C_VEL
LIN {X 0,Y 594.248,Z 681.238,A -85,B 0,C 180,E1 -1081.355,E2 -1081.355} C_VEL
LIN {X 0,Y 594.226,Z 678.915,A -85,B 0,C 180,E1 -1082.712,E2 -1082.712} C_VEL
LIN {X 0,Y 594.289,Z 676.043,A -85,B 0,C 180,E1 -1083.729,E2 -1083.729} C_VEL
LIN {X 0,Y 594.242,Z 672.143,A -85,B 0,C 180,E1 -1084.749,E2 -1084.749} C_VEL
LIN {X 0,Y 594.299,Z 667.105,A -85,B 0,C 180,E1 -1085.769,E2 -1085.769} C_VEL
LIN {X 0,Y 594.316,Z 660.765,A -85,B 0,C 180,E1 -1086.791,E2 -1086.791} C_VEL
LIN {X 0,Y 594.347,Z 652.875,A -85,B 0,C 180,E1 -1087.816,E2 -1087.816} C_VEL
LIN {X 0,Y 594.381,Z 643.023,A -85,B 0,C 180,E1 -1088.842,E2 -1088.842} C_VEL
LIN {X 0,Y 594.432,Z 632.682,A -85,B 0,C 180,E1 -1089.699,E2 -1089.699} C_VEL
LIN {X 0,Y 594.489,Z 622.488,A -85,B 0,C 180,E1 -1090.386,E2 -1090.386} C_VEL
LIN {X 0,Y 594.555,Z 610.204,A -85,B 0,C 180,E1 -1091.043,E2 -1091.043} C_VEL
LIN {X 0,Y 594.578,Z 597.444,A -85,B 0,C 180,E1 -1091.55,E2 -1091.55} C_VEL
LIN {X 0,Y 594.65,Z 584.484,A -85,B 0,C 180,E1 -1091.915,E2 -1091.915} C_VEL
LIN {X 0,Y 594.68,Z 572.209,A -85,B 0,C 180,E1 -1092.131,E2 -1092.131} C_VEL
LIN {X 0,Y 594.565,Z 470.71,A -85,B 0,C 180,E1 -1093.364,E2 -1093.364} C_VEL
LIN {X 0,Y 594.4,Z 469.624,A -85,B 0,C 180,E1 -1093.395,E2 -1093.395} C_VEL
LIN {X 0,Y 594.524,Z 449.393,A -85,B 0,C 180,E1 -1096.129,E2 -1096.129} C_VEL
LIN {X 0,Y 594.631,Z 427.729,A -85,B 0,C 180,E1 -1099.098,E2 -1099.098} C_VEL
LIN {X 0,Y 594.756,Z 406.664,A -85,B 0,C 180,E1 -1102.035,E2 -1102.035} C_VEL
LIN {X 0,Y 594.668,Z 401.252,A -85,B 0,C 180,E1 -1102.804,E2 -1102.804} C_VEL
LIN {X 0,Y 594.349,Z 399.451,A -85,B 0,C 180,E1 -1103.106,E2 -1103.106} C_VEL
LIN {X 0,Y 594.365,Z 399.45,A -85,B 0,C 180,E1 -1105.945,E2 -1105.945} C_VEL
LIN {X 0,Y 594.373,Z 399.444,A -85,B 0,C 180,E1 -1108.999,E2 -1108.999} C_VEL
LIN {X 0,Y 594.375,Z 399.45,A -85,B 0,C 180,E1 -1111.642,E2 -1111.642} C_VEL
LIN {X 0,Y 594.371,Z 399.443,A -85,B 0,C 180,E1 -1114.581,E2 -1114.581} C_VEL
LIN {X 0,Y 594.391,Z 399.445,A -85,B 0,C 180,E1 -1117.608,E2 -1117.608} C_VEL
LIN {X 0,Y 594.368,Z 399.444,A -85,B 0,C 180,E1 -1120.567,E2 -1120.567} C_VEL
LIN {X 0,Y 594.369,Z 399.449,A -85,B 0,C 180,E1 -1123.299,E2 -1123.299} C_VEL
LIN {X 0,Y 594.371,Z 399.443,A -85,B 0,C 180,E1 -1126.16,E2 -1126.16} C_VEL
LIN {X 0,Y 594.383,Z 399.445,A -85,B 0,C 180,E1 -1128.536,E2 -1128.536} C_VEL
LIN {X 0,Y 594.375,Z 399.444,A -85,B 0,C 180,E1 -1131.297,E2 -1131.297} C_VEL
LIN {X 0,Y 594.351,Z 399.445,A -85,B 0,C 180,E1 -1133.755,E2 -1133.755} C_VEL
LIN {X 0,Y 594.38,Z 399.446,A -85,B 0,C 180,E1 -1136.239,E2 -1136.239} C_VEL
LIN {X 0,Y 594.365,Z 399.45,A -85,B 0,C 180,E1 -1138.649,E2 -1138.649} C_VEL
LIN {X 0,Y 594.374,Z 399.444,A -85,B 0,C 180,E1 -1141.044,E2 -1141.044} C_VEL
LIN {X 0,Y 594.367,Z 399.45,A -85,B 0,C 180,E1 -1144.055,E2 -1144.055} C_VEL
LIN {X 0,Y 594.368,Z 399.477,A -85,B 0,C 180,E1 -1144.806,E2 -1144.806} C_VEL
LIN {X 0,Y 594.988,Z 404.366,A -85,B 0,C 180,E1 -1145.44,E2 -1145.44} C_VEL
LIN {X 0,Y 594.82,Z 426.573,A -85,B 0,C 180,E1 -1148.15,E2 -1148.15} C_VEL
LIN {X 0,Y 594.724,Z 447.647,A -85,B 0,C 180,E1 -1150.678,E2 -1150.678} C_VEL
LIN {X 0,Y 594.557,Z 471.732,A -85,B 0,C 180,E1 -1153.519,E2 -1153.519} C_VEL
LIN {X 0,Y 594.468,Z 495.817,A -85,B 0,C 180,E1 -1156.323,E2 -1156.323} C_VEL
LIN {X 0,Y 594.426,Z 498.64,A -85,B 0,C 180,E1 -1156.649,E2 -1156.649} C_VEL
LIN {X 0,Y 594.728,Z 505.502,A -85,B 0,C 180,E1 -1156.743,E2 -1156.743} C_VEL
LIN {X 0,Y 594.654,Z 607.943,A -85,B 0,C 180,E1 -1157.999,E2 -1157.999} C_VEL
LIN {X 0,Y 594.626,Z 621.215,A -85,B 0,C 180,E1 -1158.301,E2 -1158.301} C_VEL
LIN {X 0,Y 594.588,Z 634.287,A -85,B 0,C 180,E1 -1158.746,E2 -1158.746} C_VEL
LIN {X 0,Y 594.532,Z 645.631,A -85,B 0,C 180,E1 -1159.27,E2 -1159.27} C_VEL
LIN {X 0,Y 594.472,Z 657.199,A -85,B 0,C 180,E1 -1159.957,E2 -1159.957} C_VEL
LIN {X 0,Y 594.414,Z 667.596,A -85,B 0,C 180,E1 -1160.73,E2 -1160.73} C_VEL
LIN {X 0,Y 594.383,Z 676.112,A -85,B 0,C 180,E1 -1161.5,E2 -1161.5} C_VEL
LIN {X 0,Y 594.347,Z 683.96,A -85,B 0,C 180,E1 -1162.355,E2 -1162.355} C_VEL
LIN {X 0,Y 594.283,Z 691.812,A -85,B 0,C 180,E1 -1163.408,E2 -1163.408} C_VEL
LIN {X 0,Y 594.289,Z 698.68,A -85,B 0,C 180,E1 -1164.571,E2 -1164.571} C_VEL
LIN {X 0,Y 594.27,Z 703.371,A -85,B 0,C 180,E1 -1165.591,E2 -1165.591} C_VEL
LIN {X 0,Y 594.267,Z 706.956,A -85,B 0,C 180,E1 -1166.61,E2 -1166.61} C_VEL
LIN {X 0,Y 594.226,Z 708.809,A -85,B 0,C 180,E1 -1167.288,E2 -1167.288} C_VEL
LIN {X 0,Y 594.241,Z 710.201,A -85,B 0,C 180,E1 -1167.967,E2 -1167.967} C_VEL
LIN {X 0,Y 594.239,Z 711.784,A -85,B 0,C 180,E1 -1169.322,E2 -1169.322} C_VEL
LIN {X 0,Y 594.236,Z 712,A -85,B 0,C 180,E1 -1170,E2 -1170} C_VEL
LIN {X 0,Y 594.247,Z 711.185,A -85,B 0,C 180,E1 -1171.355,E2 -1171.355} C_VEL
LIN {X 0,Y 594.241,Z 710.202,A -85,B 0,C 180,E1 -1172.033,E2 -1172.033} C_VEL
LIN {X 0,Y 594.226,Z 708.809,A -85,B 0,C 180,E1 -1172.712,E2 -1172.712} C_VEL
LIN {X 0,Y 594.289,Z 705.896,A -85,B 0,C 180,E1 -1173.729,E2 -1173.729} C_VEL
LIN {X 0,Y 594.241,Z 701.95,A -85,B 0,C 180,E1 -1174.749,E2 -1174.749} C_VEL
LIN {X 0,Y 594.304,Z 695.877,A -85,B 0,C 180,E1 -1175.939,E2 -1175.939} C_VEL
LIN {X 0,Y 594.308,Z 689.236,A -85,B 0,C 180,E1 -1176.962,E2 -1176.962} C_VEL
LIN {X 0,Y 594.359,Z 680.989,A -85,B 0,C 180,E1 -1177.986,E2 -1177.986} C_VEL
LIN {X 0,Y 594.382,Z 672.537,A -85,B 0,C 180,E1 -1178.842,E2 -1178.842} C_VEL
LIN {X 0,Y 594.431,Z 662.093,A -85,B 0,C 180,E1 -1179.699,E2 -1179.699} C_VEL
LIN {X 0,Y 594.489,Z 651.758,A -85,B 0,C 180,E1 -1180.386,E2 -1180.386} C_VEL
LIN {X 0,Y 594.559,Z 640.712,A -85,B 0,C 180,E1 -1180.974,E2 -1180.974} C_VEL
LIN {X 0,Y 594.573,Z 628.706,A -85,B 0,C 180,E1 -1181.464,E2 -1181.464} C_VEL
LIN {X 0,Y 594.607,Z 615.348,A -85,B 0,C 180,E1 -1181.851,E2 -1181.851} C_VEL
LIN {X 0,Y 594.674,Z 602.079,A -85,B 0,C 180,E1 -1182.088,E2 -1182.088} C_VEL
LIN {X 0,Y 594.637,Z 500.136,A -85,B 0,C 180,E1 -1183.325,E2 -1183.325} C_VEL
LIN {X 0,Y 594.439,Z 498.452,A -85,B 0,C 180,E1 -1183.373,E2 -1183.373} C_VEL
LIN {X 0,Y 594.568,Z 473.238,A -85,B 0,C 180,E1 -1186.304,E2 -1186.304} C_VEL
LIN {X 0,Y 594.711,Z 449.457,A -85,B 0,C 180,E1 -1189.107,E2 -1189.107} C_VEL
LIN {X 0,Y 594.82,Z 426.573,A -85,B 0,C 180,E1 -1191.85,E2 -1191.85} C_VEL
LIN {X 0,Y 594.986,Z 404.37,A -85,B 0,C 180,E1 -1194.559,E2 -1194.559} C_VEL
LIN {X 0,Y 594.36,Z 399.451,A -85,B 0,C 180,E1 -1195.217,E2 -1195.217} C_VEL
LIN {X 0,Y 594.355,Z 399.447,A -85,B 0,C 180,E1 -1198.228,E2 -1198.228} C_VEL
LIN {X 0,Y 594.365,Z 399.443,A -85,B 0,C 180,E1 -1200.561,E2 -1200.561} C_VEL
LIN {X 0,Y 594.375,Z 399.443,A -85,B 0,C 180,E1 -1202.951,E2 -1202.951} C_VEL
LIN {X 0,Y 594.328,Z 399.456,A -85,B 0,C 180,E1 -1205.411,E2 -1205.411} C_VEL
LIN {X 0,Y 594.382,Z 399.443,A -85,B 0,C 180,E1 -1207.941,E2 -1207.941} C_VEL
LIN {X 0,Y 594.373,Z 399.444,A -85,B 0,C 180,E1 -1210.821,E2 -1210.821} C_VEL
LIN {X 0,Y 594.364,Z 399.445,A -85,B 0,C 180,E1 -1213.839,E2 -1213.839} C_VEL
LIN {X 0,Y 594.368,Z 399.445,A -85,B 0,C 180,E1 -1216.7,E2 -1216.7} C_VEL
LIN {X 0,Y 594.372,Z 399.447,A -85,B 0,C 180,E1 -1219.433,E2 -1219.433} C_VEL
LIN {X 0,Y 594.392,Z 399.441,A -85,B 0,C 180,E1 -1222.392,E2 -1222.392} C_VEL
LIN {X 0,Y 594.382,Z 399.444,A -85,B 0,C 180,E1 -1225.42,E2 -1225.42} C_VEL
LIN {X 0,Y 594.379,Z 399.443,A -85,B 0,C 180,E1 -1228.358,E2 -1228.358} C_VEL
LIN {X 0,Y 594.38,Z 399.448,A -85,B 0,C 180,E1 -1231.043,E2 -1231.043} C_VEL
LIN {X 0,Y 594.382,Z 399.443,A -85,B 0,C 180,E1 -1233.3,E2 -1233.3} C_VEL
LIN {X 0,Y 594.39,Z 399.444,A -85,B 0,C 180,E1 -1236.296,E2 -1236.296} C_VEL
LIN {X 0,Y 594.39,Z 399.442,A -85,B 0,C 180,E1 -1239.224,E2 -1239.224} C_VEL
LIN {X 0,Y 594.343,Z 399.449,A -85,B 0,C 180,E1 -1242.095,E2 -1242.095} C_VEL
LIN {X 0,Y 594.356,Z 399.45,A -85,B 0,C 180,E1 -1244.219,E2 -1244.219} C_VEL
LIN {X 0,Y 594.367,Z 399.535,A -85,B 0,C 180,E1 -1246.011,E2 -1246.011} C_VEL
LIN {X 0,Y 594.348,Z 402.866,A -85,B 0,C 180,E1 -1246.734,E2 -1246.734} C_VEL
LIN {X 0,Y 594.771,Z 407.168,A -85,B 0,C 180,E1 -1246.809,E2 -1246.809} C_VEL
LIN {X 0,Y 594.671,Z 507.758,A -85,B 0,C 180,E1 -1248.042,E2 -1248.042} C_VEL
LIN {X 0,Y 594.622,Z 521.181,A -85,B 0,C 180,E1 -1248.344,E2 -1248.344} C_VEL
LIN {X 0,Y 594.565,Z 533.055,A -85,B 0,C 180,E1 -1248.743,E2 -1248.743} C_VEL
LIN {X 0,Y 594.531,Z 544.721,A -85,B 0,C 180,E1 -1249.27,E2 -1249.27} C_VEL
LIN {X 0,Y 594.483,Z 556.539,A -85,B 0,C 180,E1 -1249.958,E2 -1249.958} C_VEL
LIN {X 0,Y 594.406,Z 568.097,A -85,B 0,C 180,E1 -1250.815,E2 -1250.815} C_VEL
LIN {X 0,Y 594.373,Z 577.351,A -85,B 0,C 180,E1 -1251.672,E2 -1251.672} C_VEL
LIN {X 0,Y 594.317,Z 586.337,A -85,B 0,C 180,E1 -1252.697,E2 -1252.697} C_VEL
LIN {X 0,Y 594.285,Z 592.86,A -85,B 0,C 180,E1 -1253.612,E2 -1253.612} C_VEL
LIN {X 0,Y 594.289,Z 598.446,A -85,B 0,C 180,E1 -1254.571,E2 -1254.571} C_VEL
LIN {X 0,Y 594.27,Z 603.184,A -85,B 0,C 180,E1 -1255.591,E2 -1255.591} C_VEL
LIN {X 0,Y 594.267,Z 606.811,A -85,B 0,C 180,E1 -1256.61,E2 -1256.61} C_VEL
LIN {X 0,Y 594.225,Z 608.698,A -85,B 0,C 180,E1 -1257.288,E2 -1257.288} C_VEL
LIN {X 0,Y 594.241,Z 610.132,A -85,B 0,C 180,E1 -1257.967,E2 -1257.967} C_VEL
LIN {X 0,Y 594.24,Z 611.755,A -85,B 0,C 180,E1 -1259.322,E2 -1259.322} C_VEL
LIN {X 0,Y 594.236,Z 611.996,A -85,B 0,C 180,E1 -1260,E2 -1260} C_VEL
LIN {X 0,Y 594.239,Z 611.816,A -85,B 0,C 180,E1 -1260.678,E2 -1260.678} C_VEL
LIN {X 0,Y 594.242,Z 610.278,A -85,B 0,C 180,E1 -1262.033,E2 -1262.033} C_VEL
LIN {X 0,Y 594.226,Z 608.906,A -85,B 0,C 180,E1 -1262.712,E2 -1262.712} C_VEL
LIN {X 0,Y 594.289,Z 606.034,A -85,B 0,C 180,E1 -1263.729,E2 -1263.729} C_VEL
LIN {X 0,Y 594.242,Z 602.14,A -85,B 0,C 180,E1 -1264.749,E2 -1264.749} C_VEL
LIN {X 0,Y 594.299,Z 597.112,A -85,B 0,C 180,E1 -1265.769,E2 -1265.769} C_VEL
LIN {X 0,Y 594.316,Z 590.773,A -85,B 0,C 180,E1 -1266.791,E2 -1266.791} C_VEL
LIN {X 0,Y 594.347,Z 582.867,A -85,B 0,C 180,E1 -1267.816,E2 -1267.816} C_VEL
LIN {X 0,Y 594.381,Z 573.025,A -85,B 0,C 180,E1 -1268.842,E2 -1268.842} C_VEL
LIN {X 0,Y 594.432,Z 562.683,A -85,B 0,C 180,E1 -1269.699,E2 -1269.699} C_VEL
LIN {X 0,Y 594.489,Z 552.471,A -85,B 0,C 180,E1 -1270.386,E2 -1270.386} C_VEL
LIN {X 0,Y 594.561,Z 540.598,A -85,B 0,C 180,E1 -1271.024,E2 -1271.024} C_VEL
LIN {X 0,Y 594.585,Z 528.714,A -85,B 0,C 180,E1 -1271.508,E2 -1271.508} C_VEL
LIN {X 0,Y 594.627,Z 518.731,A -85,B 0,C 180,E1 -1271.814,E2 -1271.814} C_VEL
LIN {X 0,Y 594.112,Z 513.032,A -85,B 0,C 180,E1 -1271.96,E2 -1271.96} C_VEL
LIN {X 0,Y 588.898,Z 496.363,A -85,B 0,C 180,E1 -1272.326,E2 -1272.326} C_VEL
LIN {X 0,Y 587.866,Z 490.617,A -85,B 0,C 180,E1 -1272.416,E2 -1272.416} C_VEL
LIN {X 0,Y 587.793,Z 488.665,A -85,B 0,C 180,E1 -1272.441,E2 -1272.441} C_VEL
LIN {X 0,Y 587.718,Z 405.581,A -85,B 0,C 180,E1 -1273.463,E2 -1273.463} C_VEL
LIN {X 0,Y 587.288,Z 402.877,A -85,B 0,C 180,E1 -1273.517,E2 -1273.517} C_VEL
LIN {X 0,Y 587.317,Z 400.325,A -85,B 0,C 180,E1 -1274.125,E2 -1274.125} C_VEL
LIN {X 0,Y 587.318,Z 400.322,A -85,B 0,C 180,E1 -1276.803,E2 -1276.803} C_VEL
LIN {X 0,Y 587.31,Z 400.331,A -85,B 0,C 180,E1 -1279.576,E2 -1279.576} C_VEL
LIN {X 0,Y 587.317,Z 400.325,A -85,B 0,C 180,E1 -1281.775,E2 -1281.775} C_VEL
LIN {X 0,Y 587.343,Z 400.318,A -85,B 0,C 180,E1 -1284.577,E2 -1284.577} C_VEL
LIN {X 0,Y 587.344,Z 400.32,A -85,B 0,C 180,E1 -1287.691,E2 -1287.691} C_VEL
LIN {X 0,Y 587.339,Z 400.319,A -85,B 0,C 180,E1 -1290.51,E2 -1290.51} C_VEL
LIN {X 0,Y 587.335,Z 400.322,A -85,B 0,C 180,E1 -1293.397,E2 -1293.397} C_VEL
LIN {X 0,Y 587.294,Z 400.324,A -85,B 0,C 180,E1 -1295.9,E2 -1295.9} C_VEL
LIN {X 0,Y 587.334,Z 400.321,A -85,B 0,C 180,E1 -1298.479,E2 -1298.479} C_VEL
LIN {X 0,Y 587.338,Z 400.324,A -85,B 0,C 180,E1 -1301.157,E2 -1301.157} C_VEL
LIN {X 0,Y 587.33,Z 400.32,A -85,B 0,C 180,E1 -1304.113,E2 -1304.113} C_VEL
LIN {X 0,Y 587.321,Z 400.326,A -85,B 0,C 180,E1 -1306.994,E2 -1306.994} C_VEL
LIN {X 0,Y 587.312,Z 400.321,A -85,B 0,C 180,E1 -1309.745,E2 -1309.745} C_VEL
LIN {X 0,Y 587.344,Z 400.324,A -85,B 0,C 180,E1 -1312.392,E2 -1312.392} C_VEL
LIN {X 0,Y 587.356,Z 400.317,A -85,B 0,C 180,E1 -1315.779,E2 -1315.779} C_VEL
LIN {X 0,Y 587.334,Z 400.325,A -85,B 0,C 180,E1 -1318.23,E2 -1318.23} C_VEL
LIN {X 0,Y 587.344,Z 400.321,A -85,B 0,C 180,E1 -1320.868,E2 -1320.868} C_VEL
LIN {X 0,Y 587.309,Z 400.326,A -85,B 0,C 180,E1 -1323.83,E2 -1323.83} C_VEL
LIN {X 0,Y 587.298,Z 400.33,A -85,B 0,C 180,E1 -1326.74,E2 -1326.74} C_VEL
LIN {X 0,Y 587.327,Z 400.511,A -85,B 0,C 180,E1 -1326.878,E2 -1326.878} C_VEL
LIN {X 0,Y 587.858,Z 404.736,A -85,B 0,C 180,E1 -1327.507,E2 -1327.507} C_VEL
LIN {X 0,Y 587.712,Z 425.442,A -85,B 0,C 180,E1 -1330.438,E2 -1330.438} C_VEL
LIN {X 0,Y 587.531,Z 443.331,A -85,B 0,C 180,E1 -1332.927,E2 -1332.927} C_VEL
LIN {X 0,Y 587.446,Z 464.574,A -85,B 0,C 180,E1 -1335.845,E2 -1335.845} C_VEL
LIN {X 0,Y 587.426,Z 469.605,A -85,B 0,C 180,E1 -1336.531,E2 -1336.531} C_VEL
LIN {X 0,Y 587.825,Z 473.634,A -85,B 0,C 180,E1 -1336.606,E2 -1336.606} C_VEL
LIN {X 0,Y 587.724,Z 577.716,A -85,B 0,C 180,E1 -1337.899,E2 -1337.899} C_VEL
LIN {X 0,Y 587.649,Z 590.439,A -85,B 0,C 180,E1 -1338.182,E2 -1338.182} C_VEL
LIN {X 0,Y 587.608,Z 603.775,A -85,B 0,C 180,E1 -1338.635,E2 -1338.635} C_VEL
LIN {X 0,Y 587.546,Z 614.761,A -85,B 0,C 180,E1 -1339.141,E2 -1339.141} C_VEL
LIN {X 0,Y 587.449,Z 625.198,A -85,B 0,C 180,E1 -1339.749,E2 -1339.749} C_VEL
LIN {X 0,Y 587.395,Z 634.885,A -85,B 0,C 180,E1 -1340.444,E2 -1340.444} C_VEL
LIN {X 0,Y 587.336,Z 643.865,A -85,B 0,C 180,E1 -1341.224,E2 -1341.224} C_VEL
LIN {X 0,Y 587.274,Z 653.579,A -85,B 0,C 180,E1 -1342.263,E2 -1342.263} C_VEL
LIN {X 0,Y 587.247,Z 661.819,A -85,B 0,C 180,E1 -1343.376,E2 -1343.376} C_VEL
LIN {X 0,Y 587.211,Z 668.43,A -85,B 0,C 180,E1 -1344.506,E2 -1344.506} C_VEL
LIN {X 0,Y 587.188,Z 673.165,A -85,B 0,C 180,E1 -1345.538,E2 -1345.538} C_VEL
LIN {X 0,Y 587.193,Z 676.805,A -85,B 0,C 180,E1 -1346.569,E2 -1346.569} C_VEL
LIN {X 0,Y 587.131,Z 678.691,A -85,B 0,C 180,E1 -1347.256,E2 -1347.256} C_VEL
LIN {X 0,Y 587.14,Z 680.133,A -85,B 0,C 180,E1 -1347.942,E2 -1347.942} C_VEL
LIN {X 0,Y 587.14,Z 681.755,A -85,B 0,C 180,E1 -1349.314,E2 -1349.314} C_VEL
LIN {X 0,Y 587.137,Z 681.996,A -85,B 0,C 180,E1 -1350,E2 -1350} C_VEL
LIN {X 0,Y 587.148,Z 681.233,A -85,B 0,C 180,E1 -1351.372,E2 -1351.372} C_VEL
LIN {X 0,Y 587.141,Z 680.278,A -85,B 0,C 180,E1 -1352.058,E2 -1352.058} C_VEL
LIN {X 0,Y 587.132,Z 678.891,A -85,B 0,C 180,E1 -1352.744,E2 -1352.744} C_VEL
LIN {X 0,Y 587.213,Z 676.016,A -85,B 0,C 180,E1 -1353.774,E2 -1353.774} C_VEL
LIN {X 0,Y 587.146,Z 672.117,A -85,B 0,C 180,E1 -1354.806,E2 -1354.806} C_VEL
LIN {X 0,Y 587.229,Z 667.092,A -85,B 0,C 180,E1 -1355.839,E2 -1355.839} C_VEL
LIN {X 0,Y 587.23,Z 660.782,A -85,B 0,C 180,E1 -1356.874,E2 -1356.874} C_VEL
LIN {X 0,Y 587.288,Z 652.865,A -85,B 0,C 180,E1 -1357.91,E2 -1357.91} C_VEL
LIN {X 0,Y 587.324,Z 644.794,A -85,B 0,C 180,E1 -1358.776,E2 -1358.776} C_VEL
LIN {X 0,Y 587.387,Z 634.924,A -85,B 0,C 180,E1 -1359.643,E2 -1359.643} C_VEL
LIN {X 0,Y 587.469,Z 625.242,A -85,B 0,C 180,E1 -1360.338,E2 -1360.338} C_VEL
LIN {X 0,Y 587.577,Z 613.093,A -85,B 0,C 180,E1 -1361.033,E2 -1361.033} C_VEL
LIN {X 0,Y 587.632,Z 600.11,A -85,B 0,C 180,E1 -1361.596,E2 -1361.596} C_VEL
LIN {X 0,Y 587.68,Z 588.021,A -85,B 0,C 180,E1 -1361.971,E2 -1361.971} C_VEL
LIN {X 0,Y 587.737,Z 576.54,A -85,B 0,C 180,E1 -1362.21,E2 -1362.21} C_VEL
LIN {X 0,Y 587.723,Z 471.901,A -85,B 0,C 180,E1 -1363.508,E2 -1363.508} C_VEL
LIN {X 0,Y 587.391,Z 469.619,A -85,B 0,C 180,E1 -1363.558,E2 -1363.558} C_VEL
LIN {X 0,Y 587.544,Z 449.389,A -85,B 0,C 180,E1 -1366.326,E2 -1366.326} C_VEL
LIN {X 0,Y 587.679,Z 428.074,A -85,B 0,C 180,E1 -1369.284,E2 -1369.284} C_VEL
LIN {X 0,Y 587.851,Z 407.954,A -85,B 0,C 180,E1 -1372.123,E2 -1372.123} C_VEL
LIN {X 0,Y 587.572,Z 401.622,A -85,B 0,C 180,E1 -1373.042,E2 -1373.042} C_VEL
LIN {X 0,Y 587.293,Z 400.331,A -85,B 0,C 180,E1 -1373.26,E2 -1373.26} C_VEL
LIN {X 0,Y 587.307,Z 400.327,A -85,B 0,C 180,E1 -1376.17,E2 -1376.17} C_VEL
LIN {X 0,Y 587.343,Z 400.32,A -85,B 0,C 180,E1 -1379.132,E2 -1379.132} C_VEL
LIN {X 0,Y 587.342,Z 400.323,A -85,B 0,C 180,E1 -1381.835,E2 -1381.835} C_VEL
LIN {X 0,Y 587.343,Z 400.318,A -85,B 0,C 180,E1 -1384.347,E2 -1384.347} C_VEL
LIN {X 0,Y 587.345,Z 400.323,A -85,B 0,C 180,E1 -1387.608,E2 -1387.608} C_VEL
LIN {X 0,Y 587.313,Z 400.321,A -85,B 0,C 180,E1 -1390.255,E2 -1390.255} C_VEL
LIN {X 0,Y 587.318,Z 400.33,A -85,B 0,C 180,E1 -1393.118,E2 -1393.118} C_VEL
LIN {X 0,Y 587.326,Z 400.32,A -85,B 0,C 180,E1 -1396.05,E2 -1396.05} C_VEL
LIN {X 0,Y 587.339,Z 400.328,A -85,B 0,C 180,E1 -1398.925,E2 -1398.925} C_VEL
LIN {X 0,Y 587.328,Z 400.32,A -85,B 0,C 180,E1 -1401.52,E2 -1401.52} C_VEL
LIN {X 0,Y 587.297,Z 400.328,A -85,B 0,C 180,E1 -1404.463,E2 -1404.463} C_VEL
LIN {X 0,Y 587.34,Z 400.323,A -85,B 0,C 180,E1 -1406.889,E2 -1406.889} C_VEL
LIN {X 0,Y 587.324,Z 400.32,A -85,B 0,C 180,E1 -1409.493,E2 -1409.493} C_VEL
LIN {X 0,Y 587.303,Z 400.329,A -85,B 0,C 180,E1 -1412.18,E2 -1412.18} C_VEL
LIN {X 0,Y 587.325,Z 400.329,A -85,B 0,C 180,E1 -1414.483,E2 -1414.483} C_VEL
LIN {X 0,Y 587.328,Z 400.509,A -85,B 0,C 180,E1 -1416.878,E2 -1416.878} C_VEL
LIN {X 0,Y 587.847,Z 404.736,A -85,B 0,C 180,E1 -1417.507,E2 -1417.507} C_VEL
LIN {X 0,Y 587.712,Z 425.441,A -85,B 0,C 180,E1 -1420.438,E2 -1420.438} C_VEL
LIN {X 0,Y 587.531,Z 443.33,A -85,B 0,C 180,E1 -1422.926,E2 -1422.926} C_VEL
LIN {X 0,Y 587.457,Z 464.541,A -85,B 0,C 180,E1 -1425.841,E2 -1425.841} C_VEL
LIN {X 0,Y 587.426,Z 469.605,A -85,B 0,C 180,E1 -1426.531,E2 -1426.531} C_VEL
LIN {X 0,Y 587.825,Z 473.632,A -85,B 0,C 180,E1 -1426.606,E2 -1426.606} C_VEL
LIN {X 0,Y 587.724,Z 577.739,A -85,B 0,C 180,E1 -1427.899,E2 -1427.899} C_VEL
LIN {X 0,Y 587.649,Z 590.445,A -85,B 0,C 180,E1 -1428.182,E2 -1428.182} C_VEL
LIN {X 0,Y 587.633,Z 603.86,A -85,B 0,C 180,E1 -1428.639,E2 -1428.639} C_VEL
LIN {X 0,Y 587.548,Z 614.724,A -85,B 0,C 180,E1 -1429.141,E2 -1429.141} C_VEL
LIN {X 0,Y 587.473,Z 626.548,A -85,B 0,C 180,E1 -1429.837,E2 -1429.837} C_VEL
LIN {X 0,Y 587.384,Z 638.108,A -85,B 0,C 180,E1 -1430.704,E2 -1430.704} C_VEL
LIN {X 0,Y 587.341,Z 647.337,A -85,B 0,C 180,E1 -1431.571,E2 -1431.571} C_VEL
LIN {X 0,Y 587.272,Z 654.964,A -85,B 0,C 180,E1 -1432.436,E2 -1432.436} C_VEL
LIN {X 0,Y 587.247,Z 661.825,A -85,B 0,C 180,E1 -1433.376,E2 -1433.376} C_VEL
LIN {X 0,Y 587.211,Z 668.448,A -85,B 0,C 180,E1 -1434.506,E2 -1434.506} C_VEL
LIN {X 0,Y 587.188,Z 673.192,A -85,B 0,C 180,E1 -1435.538,E2 -1435.538} C_VEL
LIN {X 0,Y 587.193,Z 676.825,A -85,B 0,C 180,E1 -1436.569,E2 -1436.569} C_VEL
LIN {X 0,Y 587.131,Z 678.683,A -85,B 0,C 180,E1 -1437.256,E2 -1437.256} C_VEL
LIN {X 0,Y 587.14,Z 680.109,A -85,B 0,C 180,E1 -1437.942,E2 -1437.942} C_VEL
LIN {X 0,Y 587.146,Z 681.136,A -85,B 0,C 180,E1 -1438.628,E2 -1438.628} C_VEL
LIN {X 0,Y 587.14,Z 681.752,A -85,B 0,C 180,E1 -1439.314,E2 -1439.314} C_VEL
LIN {X 0,Y 587.14,Z 681.813,A -85,B 0,C 180,E1 -1440.686,E2 -1440.686} C_VEL
LIN {X 0,Y 587.148,Z 681.239,A -85,B 0,C 180,E1 -1441.372,E2 -1441.372} C_VEL
LIN {X 0,Y 587.133,Z 678.912,A -85,B 0,C 180,E1 -1442.744,E2 -1442.744} C_VEL
LIN {X 0,Y 587.213,Z 676.041,A -85,B 0,C 180,E1 -1443.774,E2 -1443.774} C_VEL
LIN {X 0,Y 587.147,Z 672.14,A -85,B 0,C 180,E1 -1444.806,E2 -1444.806} C_VEL
LIN {X 0,Y 587.229,Z 667.094,A -85,B 0,C 180,E1 -1445.839,E2 -1445.839} C_VEL
LIN {X 0,Y 587.229,Z 660.752,A -85,B 0,C 180,E1 -1446.874,E2 -1446.874} C_VEL
LIN {X 0,Y 587.288,Z 652.873,A -85,B 0,C 180,E1 -1447.91,E2 -1447.91} C_VEL
LIN {X 0,Y 587.343,Z 643.014,A -85,B 0,C 180,E1 -1448.949,E2 -1448.949} C_VEL
LIN {X 0,Y 587.398,Z 633.818,A -85,B 0,C 180,E1 -1449.73,E2 -1449.73} C_VEL
LIN {X 0,Y 587.485,Z 623.876,A -85,B 0,C 180,E1 -1450.424,E2 -1450.424} C_VEL
LIN {X 0,Y 587.584,Z 611.652,A -85,B 0,C 180,E1 -1451.104,E2 -1451.104} C_VEL
LIN {X 0,Y 587.608,Z 598.869,A -85,B 0,C 180,E1 -1451.64,E2 -1451.64} C_VEL
LIN {X 0,Y 587.673,Z 586.276,A -85,B 0,C 180,E1 -1452.015,E2 -1452.015} C_VEL
LIN {X 0,Y 587.717,Z 573.681,A -85,B 0,C 180,E1 -1452.255,E2 -1452.255} C_VEL
LIN {X 0,Y 587.723,Z 471.905,A -85,B 0,C 180,E1 -1453.508,E2 -1453.508} C_VEL
LIN {X 0,Y 587.391,Z 469.619,A -85,B 0,C 180,E1 -1453.558,E2 -1453.558} C_VEL
LIN {X 0,Y 587.544,Z 449.389,A -85,B 0,C 180,E1 -1456.326,E2 -1456.326} C_VEL
LIN {X 0,Y 587.678,Z 428.074,A -85,B 0,C 180,E1 -1459.284,E2 -1459.284} C_VEL
LIN {X 0,Y 587.851,Z 407.955,A -85,B 0,C 180,E1 -1462.123,E2 -1462.123} C_VEL
LIN {X 0,Y 587.573,Z 401.619,A -85,B 0,C 180,E1 -1463.042,E2 -1463.042} C_VEL
LIN {X 0,Y 587.293,Z 400.331,A -85,B 0,C 180,E1 -1463.26,E2 -1463.26} C_VEL
LIN {X 0,Y 587.307,Z 400.326,A -85,B 0,C 180,E1 -1466.17,E2 -1466.17} C_VEL
LIN {X 0,Y 587.343,Z 400.321,A -85,B 0,C 180,E1 -1469.132,E2 -1469.132} C_VEL
LIN {X 0,Y 587.342,Z 400.323,A -85,B 0,C 180,E1 -1471.835,E2 -1471.835} C_VEL
LIN {X 0,Y 587.344,Z 400.318,A -85,B 0,C 180,E1 -1474.347,E2 -1474.347} C_VEL
LIN {X 0,Y 587.346,Z 400.322,A -85,B 0,C 180,E1 -1477.608,E2 -1477.608} C_VEL
LIN {X 0,Y 587.314,Z 400.322,A -85,B 0,C 180,E1 -1480.255,E2 -1480.255} C_VEL
LIN {X 0,Y 587.318,Z 400.33,A -85,B 0,C 180,E1 -1483.118,E2 -1483.118} C_VEL
LIN {X 0,Y 587.326,Z 400.32,A -85,B 0,C 180,E1 -1486.05,E2 -1486.05} C_VEL
LIN {X 0,Y 587.338,Z 400.327,A -85,B 0,C 180,E1 -1488.925,E2 -1488.925} C_VEL
LIN {X 0,Y 587.324,Z 400.321,A -85,B 0,C 180,E1 -1491.52,E2 -1491.52} C_VEL
LIN {X 0,Y 587.291,Z 400.326,A -85,B 0,C 180,E1 -1494.1,E2 -1494.1} C_VEL
LIN {X 0,Y 587.336,Z 400.328,A -85,B 0,C 180,E1 -1496.603,E2 -1496.603} C_VEL
LIN {X 0,Y 587.322,Z 400.321,A -85,B 0,C 180,E1 -1499.493,E2 -1499.493} C_VEL
LIN {X 0,Y 587.301,Z 400.331,A -85,B 0,C 180,E1 -1502.18,E2 -1502.18} C_VEL
LIN {X 0,Y 587.317,Z 400.419,A -85,B 0,C 180,E1 -1504.601,E2 -1504.601} C_VEL
LIN {X 0,Y 588.166,Z 405.498,A -85,B 0,C 180,E1 -1505.278,E2 -1505.278} C_VEL
LIN {X 0,Y 587.952,Z 426.573,A -85,B 0,C 180,E1 -1507.881,E2 -1507.881} C_VEL
LIN {X 0,Y 587.802,Z 448.738,A -85,B 0,C 180,E1 -1510.572,E2 -1510.572} C_VEL
LIN {X 0,Y 587.603,Z 471.732,A -85,B 0,C 180,E1 -1513.318,E2 -1513.318} C_VEL
LIN {X 0,Y 587.455,Z 495.817,A -85,B 0,C 180,E1 -1516.157,E2 -1516.157} C_VEL
LIN {X 0,Y 587.442,Z 498.64,A -85,B 0,C 180,E1 -1516.487,E2 -1516.487} C_VEL
LIN {X 0,Y 587.839,Z 505.502,A -85,B 0,C 180,E1 -1516.584,E2 -1516.584} C_VEL
LIN {X 0,Y 587.716,Z 607.943,A -85,B 0,C 180,E1 -1517.855,E2 -1517.855} C_VEL
LIN {X 0,Y 587.677,Z 621.216,A -85,B 0,C 180,E1 -1518.16,E2 -1518.16} C_VEL
LIN {X 0,Y 587.594,Z 633.623,A -85,B 0,C 180,E1 -1518.584,E2 -1518.584} C_VEL
LIN {X 0,Y 587.55,Z 645.63,A -85,B 0,C 180,E1 -1519.141,E2 -1519.141} C_VEL
LIN {X 0,Y 587.454,Z 657.2,A -85,B 0,C 180,E1 -1519.836,E2 -1519.836} C_VEL
LIN {X 0,Y 587.393,Z 667.597,A -85,B 0,C 180,E1 -1520.618,E2 -1520.618} C_VEL
LIN {X 0,Y 587.322,Z 676.112,A -85,B 0,C 180,E1 -1521.398,E2 -1521.398} C_VEL
LIN {X 0,Y 587.274,Z 683.96,A -85,B 0,C 180,E1 -1522.263,E2 -1522.263} C_VEL
LIN {X 0,Y 587.23,Z 690.469,A -85,B 0,C 180,E1 -1523.126,E2 -1523.126} C_VEL
LIN {X 0,Y 587.236,Z 696.866,A -85,B 0,C 180,E1 -1524.161,E2 -1524.161} C_VEL
LIN {X 0,Y 587.147,Z 701.95,A -85,B 0,C 180,E1 -1525.194,E2 -1525.194} C_VEL
LIN {X 0,Y 587.213,Z 705.896,A -85,B 0,C 180,E1 -1526.226,E2 -1526.226} C_VEL
LIN {X 0,Y 587.132,Z 708.809,A -85,B 0,C 180,E1 -1527.256,E2 -1527.256} C_VEL
LIN {X 0,Y 587.14,Z 710.2,A -85,B 0,C 180,E1 -1527.942,E2 -1527.942} C_VEL
LIN {X 0,Y 587.14,Z 711.784,A -85,B 0,C 180,E1 -1529.314,E2 -1529.314} C_VEL
LIN {X 0,Y 587.137,Z 712,A -85,B 0,C 180,E1 -1530,E2 -1530} C_VEL
LIN {X 0,Y 587.147,Z 711.185,A -85,B 0,C 180,E1 -1531.372,E2 -1531.372} C_VEL
LIN {X 0,Y 587.14,Z 710.201,A -85,B 0,C 180,E1 -1532.058,E2 -1532.058} C_VEL
LIN {X 0,Y 587.132,Z 708.81,A -85,B 0,C 180,E1 -1532.744,E2 -1532.744} C_VEL
LIN {X 0,Y 587.213,Z 705.896,A -85,B 0,C 180,E1 -1533.774,E2 -1533.774} C_VEL
LIN {X 0,Y 587.147,Z 701.949,A -85,B 0,C 180,E1 -1534.806,E2 -1534.806} C_VEL
LIN {X 0,Y 587.217,Z 695.877,A -85,B 0,C 180,E1 -1536.011,E2 -1536.011} C_VEL
LIN {X 0,Y 587.245,Z 689.236,A -85,B 0,C 180,E1 -1537.046,E2 -1537.046} C_VEL
LIN {X 0,Y 587.3,Z 680.99,A -85,B 0,C 180,E1 -1538.083,E2 -1538.083} C_VEL
LIN {X 0,Y 587.343,Z 672.537,A -85,B 0,C 180,E1 -1538.949,E2 -1538.949} C_VEL
LIN {X 0,Y 587.419,Z 662.094,A -85,B 0,C 180,E1 -1539.816,E2 -1539.816} C_VEL
LIN {X 0,Y 587.508,Z 651.757,A -85,B 0,C 180,E1 -1540.511,E2 -1540.511} C_VEL
LIN {X 0,Y 587.568,Z 639.978,A -85,B 0,C 180,E1 -1541.141,E2 -1541.141} C_VEL
LIN {X 0,Y 587.609,Z 627.595,A -85,B 0,C 180,E1 -1541.64,E2 -1541.64} C_VEL
LIN {X 0,Y 587.69,Z 614.433,A -85,B 0,C 180,E1 -1542.014,E2 -1542.014} C_VEL
LIN {X 0,Y 587.742,Z 602.079,A -85,B 0,C 180,E1 -1542.232,E2 -1542.232} C_VEL
LIN {X 0,Y 587.734,Z 500.918,A -85,B 0,C 180,E1 -1543.475,E2 -1543.475} C_VEL
LIN {X 0,Y 587.441,Z 498.452,A -85,B 0,C 180,E1 -1543.535,E2 -1543.535} C_VEL
LIN {X 0,Y 587.607,Z 473.238,A -85,B 0,C 180,E1 -1546.503,E2 -1546.503} C_VEL
LIN {X 0,Y 587.807,Z 449.812,A -85,B 0,C 180,E1 -1549.298,E2 -1549.298} C_VEL
LIN {X 0,Y 587.952,Z 426.573,A -85,B 0,C 180,E1 -1552.119,E2 -1552.119} C_VEL
LIN {X 0,Y 588.14,Z 405.312,A -85,B 0,C 180,E1 -1554.747,E2 -1554.747} C_VEL
LIN {X 0,Y 587.323,Z 400.329,A -85,B 0,C 180,E1 -1555.422,E2 -1555.422} C_VEL
LIN {X 0,Y 587.3,Z 400.332,A -85,B 0,C 180,E1 -1557.82,E2 -1557.82} C_VEL
LIN {X 0,Y 587.321,Z 400.321,A -85,B 0,C 180,E1 -1560.507,E2 -1560.507} C_VEL
LIN {X 0,Y 587.338,Z 400.322,A -85,B 0,C 180,E1 -1563.111,E2 -1563.111} C_VEL
LIN {X 0,Y 587.279,Z 400.336,A -85,B 0,C 180,E1 -1565.535,E2 -1565.535} C_VEL
LIN {X 0,Y 587.337,Z 400.322,A -85,B 0,C 180,E1 -1567.838,E2 -1567.838} C_VEL
LIN {X 0,Y 587.31,Z 400.322,A -85,B 0,C 180,E1 -1570.255,E2 -1570.255} C_VEL
LIN {X 0,Y 587.307,Z 400.329,A -85,B 0,C 180,E1 -1573.117,E2 -1573.117} C_VEL
LIN {X 0,Y 587.325,Z 400.32,A -85,B 0,C 180,E1 -1576.05,E2 -1576.05} C_VEL
LIN {X 0,Y 587.337,Z 400.324,A -85,B 0,C 180,E1 -1578.925,E2 -1578.925} C_VEL
LIN {X 0,Y 587.332,Z 400.322,A -85,B 0,C 180,E1 -1581.521,E2 -1581.521} C_VEL
LIN {X 0,Y 587.294,Z 400.324,A -85,B 0,C 180,E1 -1584.1,E2 -1584.1} C_VEL
LIN {X 0,Y 587.335,Z 400.323,A -85,B 0,C 180,E1 -1586.603,E2 -1586.603} C_VEL
LIN {X 0,Y 587.339,Z 400.32,A -85,B 0,C 180,E1 -1589.49,E2 -1589.49} C_VEL
LIN {X 0,Y 587.354,Z 400.319,A -85,B 0,C 180,E1 -1592.307,E2 -1592.307} C_VEL
LIN {X 0,Y 587.356,Z 400.318,A -85,B 0,C 180,E1 -1595.42,E2 -1595.42} C_VEL
LIN {X 0,Y 587.319,Z 400.325,A -85,B 0,C 180,E1 -1598.226,E2 -1598.226} C_VEL
LIN {X 0,Y 587.334,Z 400.321,A -85,B 0,C 180,E1 -1601.151,E2 -1601.151} C_VEL
LIN {X 0,Y 587.304,Z 400.324,A -85,B 0,C 180,E1 -1603.31,E2 -1603.31} C_VEL
LIN {X 0,Y 587.305,Z 400.479,A -85,B 0,C 180,E1 -1606.046,E2 -1606.046} C_VEL
LIN {X 0,Y 587.312,Z 402.919,A -85,B 0,C 180,E1 -1606.583,E2 -1606.583} C_VEL
LIN {X 0,Y 587.864,Z 407.214,A -85,B 0,C 180,E1 -1606.651,E2 -1606.651} C_VEL
LIN {X 0,Y 587.723,Z 507.743,A -85,B 0,C 180,E1 -1607.899,E2 -1607.899} C_VEL
LIN {X 0,Y 587.668,Z 521.21,A -85,B 0,C 180,E1 -1608.204,E2 -1608.204} C_VEL
LIN {X 0,Y 587.612,Z 533.721,A -85,B 0,C 180,E1 -1608.634,E2 -1608.634} C_VEL
LIN {X 0,Y 587.549,Z 544.715,A -85,B 0,C 180,E1 -1609.141,E2 -1609.141} C_VEL
LIN {X 0,Y 587.448,Z 555.208,A -85,B 0,C 180,E1 -1609.749,E2 -1609.749} C_VEL
LIN {X 0,Y 587.381,Z 565.996,A -85,B 0,C 180,E1 -1610.531,E2 -1610.531} C_VEL
LIN {X 0,Y 587.323,Z 575.652,A -85,B 0,C 180,E1 -1611.398,E2 -1611.398} C_VEL
LIN {X 0,Y 587.273,Z 583.552,A -85,B 0,C 180,E1 -1612.263,E2 -1612.263} C_VEL
LIN {X 0,Y 587.233,Z 590.127,A -85,B 0,C 180,E1 -1613.126,E2 -1613.126} C_VEL
LIN {X 0,Y 587.237,Z 596.606,A -85,B 0,C 180,E1 -1614.161,E2 -1614.161} C_VEL
LIN {X 0,Y 587.146,Z 601.758,A -85,B 0,C 180,E1 -1615.194,E2 -1615.194} C_VEL
LIN {X 0,Y 587.212,Z 605.747,A -85,B 0,C 180,E1 -1616.226,E2 -1616.226} C_VEL
LIN {X 0,Y 587.131,Z 608.7,A -85,B 0,C 180,E1 -1617.256,E2 -1617.256} C_VEL
LIN {X 0,Y 587.14,Z 610.133,A -85,B 0,C 180,E1 -1617.942,E2 -1617.942} C_VEL
LIN {X 0,Y 587.14,Z 611.757,A -85,B 0,C 180,E1 -1619.314,E2 -1619.314} C_VEL
LIN {X 0,Y 587.137,Z 611.996,A -85,B 0,C 180,E1 -1620,E2 -1620} C_VEL
LIN {X 0,Y 587.14,Z 611.811,A -85,B 0,C 180,E1 -1620.686,E2 -1620.686} C_VEL
LIN {X 0,Y 587.141,Z 610.279,A -85,B 0,C 180,E1 -1622.058,E2 -1622.058} C_VEL
LIN {X 0,Y 587.132,Z 608.899,A -85,B 0,C 180,E1 -1622.744,E2 -1622.744} C_VEL
LIN {X 0,Y 587.213,Z 606.03,A -85,B 0,C 180,E1 -1623.774,E2 -1623.774} C_VEL
LIN {X 0,Y 587.147,Z 602.138,A -85,B 0,C 180,E1 -1624.806,E2 -1624.806} C_VEL
LIN {X 0,Y 587.229,Z 597.111,A -85,B 0,C 180,E1 -1625.839,E2 -1625.839} C_VEL
LIN {X 0,Y 587.23,Z 590.761,A -85,B 0,C 180,E1 -1626.874,E2 -1626.874} C_VEL
LIN {X 0,Y 587.288,Z 582.86,A -85,B 0,C 180,E1 -1627.91,E2 -1627.91} C_VEL
LIN {X 0,Y 587.343,Z 573.02,A -85,B 0,C 180,E1 -1628.949,E2 -1628.949} C_VEL
LIN {X 0,Y 587.419,Z 562.67,A -85,B 0,C 180,E1 -1629.816,E2 -1629.816} C_VEL
LIN {X 0,Y 587.492,Z 552.454,A -85,B 0,C 180,E1 -1630.511,E2 -1630.511} C_VEL
LIN {X 0,Y 587.585,Z 541.401,A -85,B 0,C 180,E1 -1631.116,E2 -1631.116} C_VEL
LIN {X 0,Y 587.615,Z 528.871,A -85,B 0,C 180,E1 -1631.641,E2 -1631.641} C_VEL
LIN {X 0,Y 587.705,Z 516.246,A -85,B 0,C 180,E1 -1632.014,E2 -1632.014} C_VEL
LIN {X 0,Y 587.766,Z 503.676,A -85,B 0,C 180,E1 -1632.254,E2 -1632.254} C_VEL
LIN {X 0,Y 587.793,Z 488.665,A -85,B 0,C 180,E1 -1632.441,E2 -1632.441} C_VEL
LIN {X 0,Y 587.175,Z 482.857,A -85,B 0,C 180,E1 -1632.525,E2 -1632.525} C_VEL
LIN {X 0,Y 581.578,Z 464.168,A -85,B 0,C 180,E1 -1632.879,E2 -1632.879} C_VEL
LIN {X 0,Y 580.905,Z 458.36,A -85,B 0,C 180,E1 -1632.966,E2 -1632.966} C_VEL
LIN {X 0,Y 580.863,Z 406.654,A -85,B 0,C 180,E1 -1633.611,E2 -1633.611} C_VEL
LIN {X 0,Y 580.248,Z 402.874,A -85,B 0,C 180,E1 -1633.684,E2 -1633.684} C_VEL
LIN {X 0,Y 580.29,Z 401.201,A -85,B 0,C 180,E1 -1634.112,E2 -1634.112} C_VEL
LIN {X 0,Y 580.27,Z 401.201,A -85,B 0,C 180,E1 -1636.899,E2 -1636.899} C_VEL
LIN {X 0,Y 580.283,Z 401.202,A -85,B 0,C 180,E1 -1639.823,E2 -1639.823} C_VEL
LIN {X 0,Y 580.259,Z 401.201,A -85,B 0,C 180,E1 -1642.053,E2 -1642.053} C_VEL
LIN {X 0,Y 580.29,Z 401.201,A -85,B 0,C 180,E1 -1645.081,E2 -1645.081} C_VEL
LIN {X 0,Y 580.295,Z 401.195,A -85,B 0,C 180,E1 -1648.186,E2 -1648.186} C_VEL
LIN {X 0,Y 580.287,Z 401.199,A -85,B 0,C 180,E1 -1650.694,E2 -1650.694} C_VEL
LIN {X 0,Y 580.305,Z 401.199,A -85,B 0,C 180,E1 -1653.316,E2 -1653.316} C_VEL
LIN {X 0,Y 580.248,Z 401.202,A -85,B 0,C 180,E1 -1655.756,E2 -1655.756} C_VEL
LIN {X 0,Y 580.292,Z 401.196,A -85,B 0,C 180,E1 -1658.146,E2 -1658.146} C_VEL
LIN {X 0,Y 580.301,Z 401.202,A -85,B 0,C 180,E1 -1660.843,E2 -1660.843} C_VEL
LIN {X 0,Y 580.282,Z 401.198,A -85,B 0,C 180,E1 -1663.658,E2 -1663.658} C_VEL
LIN {X 0,Y 580.285,Z 401.203,A -85,B 0,C 180,E1 -1666.609,E2 -1666.609} C_VEL
LIN {X 0,Y 580.299,Z 401.197,A -85,B 0,C 180,E1 -1669.156,E2 -1669.156} C_VEL
LIN {X 0,Y 580.289,Z 401.197,A -85,B 0,C 180,E1 -1671.928,E2 -1671.928} C_VEL
LIN {X 0,Y 580.25,Z 401.209,A -85,B 0,C 180,E1 -1674.452,E2 -1674.452} C_VEL
LIN {X 0,Y 580.29,Z 401.199,A -85,B 0,C 180,E1 -1676.975,E2 -1676.975} C_VEL
LIN {X 0,Y 580.283,Z 401.198,A -85,B 0,C 180,E1 -1679.424,E2 -1679.424} C_VEL
LIN {X 0,Y 580.255,Z 401.208,A -85,B 0,C 180,E1 -1682.15,E2 -1682.15} C_VEL
LIN {X 0,Y 580.278,Z 401.201,A -85,B 0,C 180,E1 -1684.919,E2 -1684.919} C_VEL
LIN {X 0,Y 580.268,Z 401.335,A -85,B 0,C 180,E1 -1686.7,E2 -1686.7} C_VEL
LIN {X 0,Y 580.941,Z 406.034,A -85,B 0,C 180,E1 -1687.412,E2 -1687.412} C_VEL
LIN {X 0,Y 580.771,Z 426.601,A -85,B 0,C 180,E1 -1690.358,E2 -1690.358} C_VEL
LIN {X 0,Y 580.562,Z 447.446,A -85,B 0,C 180,E1 -1693.291,E2 -1693.291} C_VEL
LIN {X 0,Y 580.399,Z 469.448,A -85,B 0,C 180,E1 -1696.342,E2 -1696.342} C_VEL
LIN {X 0,Y 580.568,Z 470.999,A -85,B 0,C 180,E1 -1696.402,E2 -1696.402} C_VEL
LIN {X 0,Y 580.933,Z 477.256,A -85,B 0,C 180,E1 -1696.489,E2 -1696.489} C_VEL
LIN {X 0,Y 580.805,Z 577.698,A -85,B 0,C 180,E1 -1697.752,E2 -1697.752} C_VEL
LIN {X 0,Y 580.706,Z 590.463,A -85,B 0,C 180,E1 -1698.038,E2 -1698.038} C_VEL
LIN {X 0,Y 580.635,Z 604.507,A -85,B 0,C 180,E1 -1698.526,E2 -1698.526} C_VEL
LIN {X 0,Y 580.533,Z 616.346,A -85,B 0,C 180,E1 -1699.096,E2 -1699.096} C_VEL
LIN {X 0,Y 580.453,Z 626.502,A -85,B 0,C 180,E1 -1699.712,E2 -1699.712} C_VEL
LIN {X 0,Y 580.344,Z 637.044,A -85,B 0,C 180,E1 -1700.503,E2 -1700.503} C_VEL
LIN {X 0,Y 580.301,Z 647.372,A -85,B 0,C 180,E1 -1701.468,E2 -1701.468} C_VEL
LIN {X 0,Y 580.2,Z 656.333,A -85,B 0,C 180,E1 -1702.518,E2 -1702.518} C_VEL
LIN {X 0,Y 580.17,Z 662.35,A -85,B 0,C 180,E1 -1703.377,E2 -1703.377} C_VEL
LIN {X 0,Y 580.139,Z 668.425,A -85,B 0,C 180,E1 -1704.438,E2 -1704.438} C_VEL
LIN {X 0,Y 580.108,Z 673.162,A -85,B 0,C 180,E1 -1705.483,E2 -1705.483} C_VEL
LIN {X 0,Y 580.123,Z 676.804,A -85,B 0,C 180,E1 -1706.527,E2 -1706.527} C_VEL
LIN {X 0,Y 580.043,Z 678.685,A -85,B 0,C 180,E1 -1707.222,E2 -1707.222} C_VEL
LIN {X 0,Y 580.039,Z 680.135,A -85,B 0,C 180,E1 -1707.917,E2 -1707.917} C_VEL
LIN {X 0,Y 580.041,Z 681.756,A -85,B 0,C 180,E1 -1709.306,E2 -1709.306} C_VEL
LIN {X 0,Y 580.038,Z 681.996,A -85,B 0,C 180,E1 -1710,E2 -1710} C_VEL
LIN {X 0,Y 580.047,Z 681.232,A -85,B 0,C 180,E1 -1711.389,E2 -1711.389} C_VEL
LIN {X 0,Y 580.04,Z 680.278,A -85,B 0,C 180,E1 -1712.083,E2 -1712.083} C_VEL
LIN {X 0,Y 580.123,Z 677.077,A -85,B 0,C 180,E1 -1713.473,E2 -1713.473} C_VEL
LIN {X 0,Y 580.108,Z 673.528,A -85,B 0,C 180,E1 -1714.517,E2 -1714.517} C_VEL
LIN {X 0,Y 580.137,Z 668.884,A -85,B 0,C 180,E1 -1715.562,E2 -1715.562} C_VEL
LIN {X 0,Y 580.137,Z 663.094,A -85,B 0,C 180,E1 -1716.594,E2 -1716.594} C_VEL
LIN {X 0,Y 580.221,Z 655.68,A -85,B 0,C 180,E1 -1717.657,E2 -1717.657} C_VEL
LIN {X 0,Y 580.259,Z 646.562,A -85,B 0,C 180,E1 -1718.708,E2 -1718.708} C_VEL
LIN {X 0,Y 580.359,Z 637.069,A -85,B 0,C 180,E1 -1719.585,E2 -1719.585} C_VEL
LIN {X 0,Y 580.453,Z 626.529,A -85,B 0,C 180,E1 -1720.376,E2 -1720.376} C_VEL
LIN {X 0,Y 580.553,Z 616.377,A -85,B 0,C 180,E1 -1720.992,E2 -1720.992} C_VEL
LIN {X 0,Y 580.638,Z 604.491,A -85,B 0,C 180,E1 -1721.564,E2 -1721.564} C_VEL
LIN {X 0,Y 580.721,Z 590.512,A -85,B 0,C 180,E1 -1722.05,E2 -1722.05} C_VEL
LIN {X 0,Y 580.806,Z 577.775,A -85,B 0,C 180,E1 -1722.336,E2 -1722.336} C_VEL
LIN {X 0,Y 580.811,Z 472.63,A -85,B 0,C 180,E1 -1723.662,E2 -1723.662} C_VEL
LIN {X 0,Y 580.398,Z 469.615,A -85,B 0,C 180,E1 -1723.725,E2 -1723.725} C_VEL
LIN {X 0,Y 580.566,Z 448.09,A -85,B 0,C 180,E1 -1726.709,E2 -1726.709} C_VEL
LIN {X 0,Y 580.772,Z 427.235,A -85,B 0,C 180,E1 -1729.641,E2 -1729.641} C_VEL
LIN {X 0,Y 580.955,Z 406.655,A -85,B 0,C 180,E1 -1732.587,E2 -1732.587} C_VEL
LIN {X 0,Y 580.331,Z 401.637,A -85,B 0,C 180,E1 -1733.343,E2 -1733.343} C_VEL
LIN {X 0,Y 580.262,Z 401.208,A -85,B 0,C 180,E1 -1733.417,E2 -1733.417} C_VEL
LIN {X 0,Y 580.26,Z 401.203,A -85,B 0,C 180,E1 -1736.327,E2 -1736.327} C_VEL
LIN {X 0,Y 580.278,Z 401.203,A -85,B 0,C 180,E1 -1739.305,E2 -1739.305} C_VEL
LIN {X 0,Y 580.297,Z 401.197,A -85,B 0,C 180,E1 -1742.201,E2 -1742.201} C_VEL
LIN {X 0,Y 580.288,Z 401.198,A -85,B 0,C 180,E1 -1744.697,E2 -1744.697} C_VEL
LIN {X 0,Y 580.291,Z 401.206,A -85,B 0,C 180,E1 -1747.269,E2 -1747.269} C_VEL
LIN {X 0,Y 580.293,Z 401.195,A -85,B 0,C 180,E1 -1750.27,E2 -1750.27} C_VEL
LIN {X 0,Y 580.28,Z 401.201,A -85,B 0,C 180,E1 -1752.706,E2 -1752.706} C_VEL
LIN {X 0,Y 580.274,Z 401.2,A -85,B 0,C 180,E1 -1755.609,E2 -1755.609} C_VEL
LIN {X 0,Y 580.284,Z 401.197,A -85,B 0,C 180,E1 -1758.231,E2 -1758.231} C_VEL
LIN {X 0,Y 580.287,Z 401.204,A -85,B 0,C 180,E1 -1760.965,E2 -1760.965} C_VEL
LIN {X 0,Y 580.252,Z 401.199,A -85,B 0,C 180,E1 -1763.595,E2 -1763.595} C_VEL
LIN {X 0,Y 580.315,Z 401.196,A -85,B 0,C 180,E1 -1766.145,E2 -1766.145} C_VEL
LIN {X 0,Y 580.27,Z 401.208,A -85,B 0,C 180,E1 -1768.614,E2 -1768.614} C_VEL
LIN {X 0,Y 580.286,Z 401.199,A -85,B 0,C 180,E1 -1771.023,E2 -1771.023} C_VEL
LIN {X 0,Y 580.264,Z 401.207,A -85,B 0,C 180,E1 -1774.149,E2 -1774.149} C_VEL
LIN {X 0,Y 580.269,Z 401.334,A -85,B 0,C 180,E1 -1776.7,E2 -1776.7} C_VEL
LIN {X 0,Y 580.931,Z 406.034,A -85,B 0,C 180,E1 -1777.412,E2 -1777.412} C_VEL
LIN {X 0,Y 580.771,Z 426.601,A -85,B 0,C 180,E1 -1780.358,E2 -1780.358} C_VEL
LIN {X 0,Y 580.563,Z 447.446,A -85,B 0,C 180,E1 -1783.291,E2 -1783.291} C_VEL
LIN {X 0,Y 580.399,Z 469.448,A -85,B 0,C 180,E1 -1786.342,E2 -1786.342} C_VEL
LIN {X 0,Y 580.568,Z 470.997,A -85,B 0,C 180,E1 -1786.402,E2 -1786.402} C_VEL
